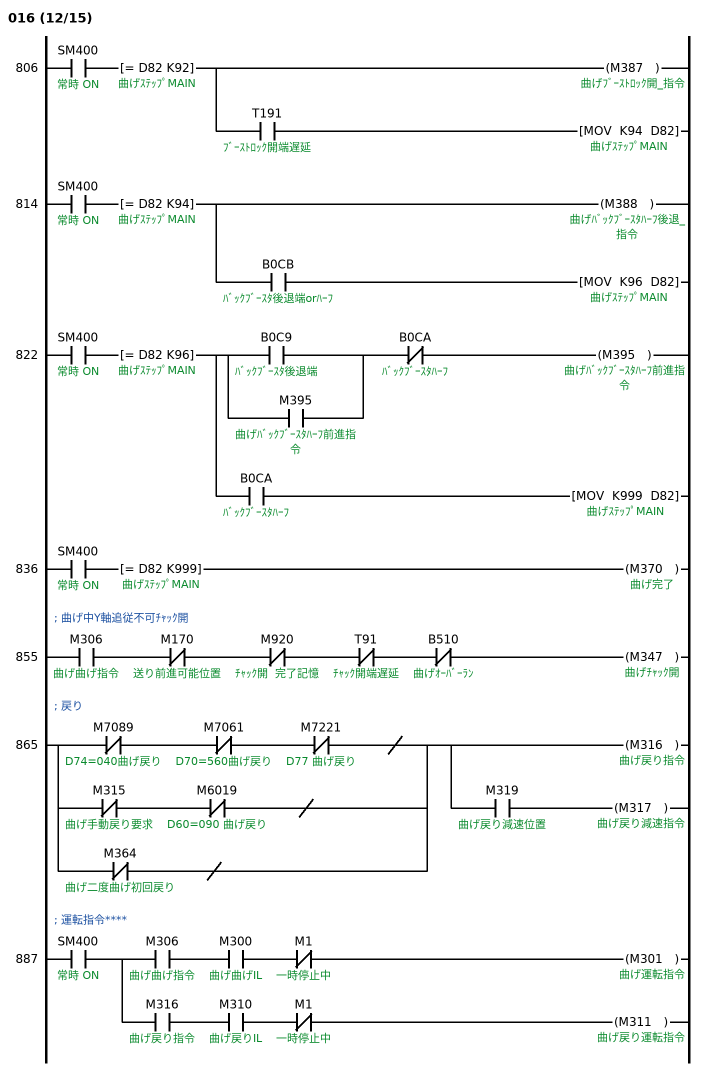
806   LD      SM400  ; 常時 ON
      AND=    D82 K92  ; 曲げｽﾃｯﾌﾟMAIN
      OUT     M387  ; 曲げﾌﾞｰｽﾄﾛｯｸ開_指令
      AND     T191  ; ﾌﾞｰｽﾄﾛｯｸ開端遅延
      MOV     K94 D82
814   LD      SM400  ; 常時 ON
      AND=    D82 K94  ; 曲げｽﾃｯﾌﾟMAIN
      OUT     M388  ; 曲げﾊﾞｯｸﾌﾞｰｽﾀﾊｰﾌ後退_指令
      AND     B0CB  ; ﾊﾞｯｸﾌﾞｰｽﾀ後退端orﾊｰﾌ
      MOV     K96 D82
822   LD      SM400  ; 常時 ON
      AND=    D82 K96  ; 曲げｽﾃｯﾌﾟMAIN
      MPS
      LD      B0C9  ; ﾊﾞｯｸﾌﾞｰｽﾀ後退端
      OR      M395  ; 曲げﾊﾞｯｸﾌﾞｰｽﾀﾊｰﾌ前進指令
      ANB
      ANI     B0CA  ; ﾊﾞｯｸﾌﾞｰｽﾀﾊｰﾌ
      OUT     M395  ; 曲げﾊﾞｯｸﾌﾞｰｽﾀﾊｰﾌ前進指令
      MPP
      AND     B0CA  ; ﾊﾞｯｸﾌﾞｰｽﾀﾊｰﾌ
      MOV     K999 D82
836   LD      SM400  ; 常時 ON
      AND=    D82 K999  ; 曲げｽﾃｯﾌﾟMAIN
      OUT     M370  ; 曲げ完了
; 曲げ中Y軸追従不可ﾁｬｯｸ開
855   LD      M306  ; 曲げ曲げ指令
      ANI     M170  ; 送り前進可能位置
      ANI     M920  ; ﾁｬｯｸ開  完了記憶
      ANI     T91  ; ﾁｬｯｸ開端遅延
      ANI     B510  ; 曲げｵｰﾊﾞｰﾗﾝ
      OUT     M347  ; 曲げﾁｬｯｸ開
; 戻り
865   LDI     M7089  ; D74=040曲げ戻り
      ANI     M7061  ; D70=560曲げ戻り
      ANI     M7221  ; D77 曲げ戻り
      INV
      LDI     M315  ; 曲げ手動戻り要求
      ANI     M6019  ; D60=090 曲げ戻り
      INV
      ORB
      LDI     M364  ; 曲げ二度曲げ初回戻り
      INV
      ORB
      OUT     M316  ; 曲げ戻り指令
      AND     M319  ; 曲げ戻り減速位置
      OUT     M317  ; 曲げ戻り減速指令
; 運転指令****
887   LD      SM400  ; 常時 ON
      MPS
      AND     M306  ; 曲げ曲げ指令
      AND     M300  ; 曲げ曲げIL
      ANI     M1  ; 一時停止中
      OUT     M301  ; 曲げ運転指令
      MPP
      AND     M316  ; 曲げ戻り指令
      AND     M310  ; 曲げ戻りIL
      ANI     M1  ; 一時停止中
      OUT     M311  ; 曲げ戻り運転指令
; 
      P1610
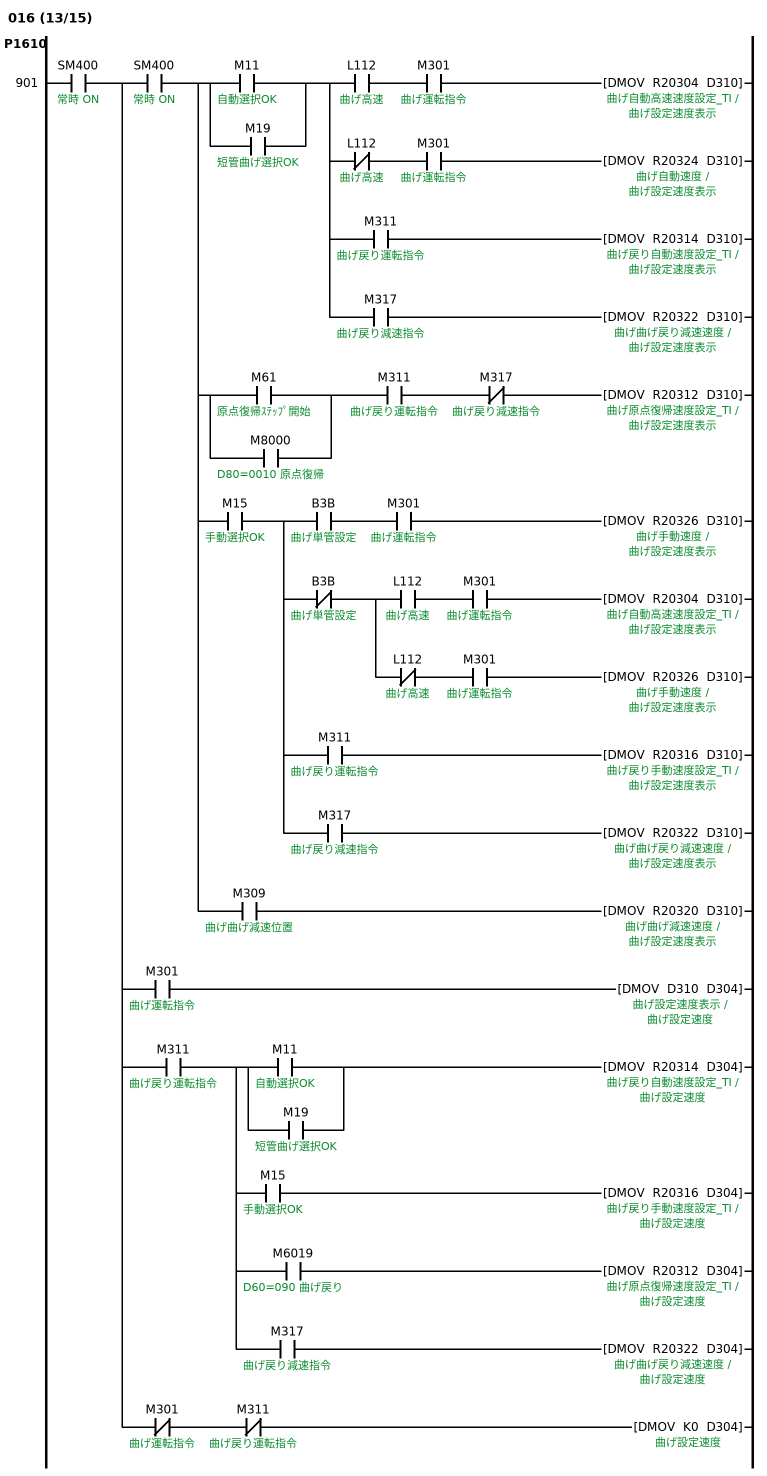
901   LD      SM400  ; 常時 ON
      MPS
      AND     SM400  ; 常時 ON
      MPS
      LD      M11  ; 自動選択OK
      OR      M19  ; 短管曲げ選択OK
      ANB
      MPS
      AND     L112  ; 曲げ高速
      AND     M301  ; 曲げ運転指令
      DMOV    R20304 D310  ; 曲げ自動高速速度設定_TI / 曲げ設定速度表示
      MRD
      ANI     L112  ; 曲げ高速
      AND     M301  ; 曲げ運転指令
      DMOV    R20324 D310  ; 曲げ自動速度
      MRD
      AND     M311  ; 曲げ戻り運転指令
      DMOV    R20314 D310  ; 曲げ戻り自動速度設定_TI
      MPP
      AND     M317  ; 曲げ戻り減速指令
      DMOV    R20322 D310  ; 曲げ曲げ戻り減速速度
      MRD
      LD      M61  ; 原点復帰ｽﾃｯﾌﾟ開始
      OR      M8000  ; D80=0010 原点復帰
      ANB
      AND     M311  ; 曲げ戻り運転指令
      ANI     M317  ; 曲げ戻り減速指令
      DMOV    R20312 D310  ; 曲げ原点復帰速度設定_TI
      MRD
      AND     M15  ; 手動選択OK
      MPS
      AND     B3B  ; 曲げ単管設定
      AND     M301  ; 曲げ運転指令
      DMOV    R20326 D310  ; 曲げ手動速度
      MRD
      ANI     B3B  ; 曲げ単管設定
      MPS
      AND     L112  ; 曲げ高速
      AND     M301  ; 曲げ運転指令
      DMOV    R20304 D310
      MPP
      ANI     L112  ; 曲げ高速
      AND     M301  ; 曲げ運転指令
      DMOV    R20326 D310
      MRD
      AND     M311  ; 曲げ戻り運転指令
      DMOV    R20316 D310  ; 曲げ戻り手動速度設定_TI
      MPP
      AND     M317  ; 曲げ戻り減速指令
      DMOV    R20322 D310
      MPP
      AND     M309  ; 曲げ曲げ減速位置
      DMOV    R20320 D310  ; 曲げ曲げ減速速度
      MRD
      AND     M301  ; 曲げ運転指令
      DMOV    D310 D304  ; 曲げ設定速度
      MRD
      AND     M311  ; 曲げ戻り運転指令
      MPS
      LD      M11  ; 自動選択OK
      OR      M19  ; 短管曲げ選択OK
      ANB
      DMOV    R20314 D304
      MRD
      AND     M15  ; 手動選択OK
      DMOV    R20316 D304
      MRD
      AND     M6019  ; D60=090 曲げ戻り
      DMOV    R20312 D304
      MPP
      AND     M317  ; 曲げ戻り減速指令
      DMOV    R20322 D304
      MPP
      ANI     M301  ; 曲げ運転指令
      ANI     M311  ; 曲げ戻り運転指令
      DMOV    K0 D304
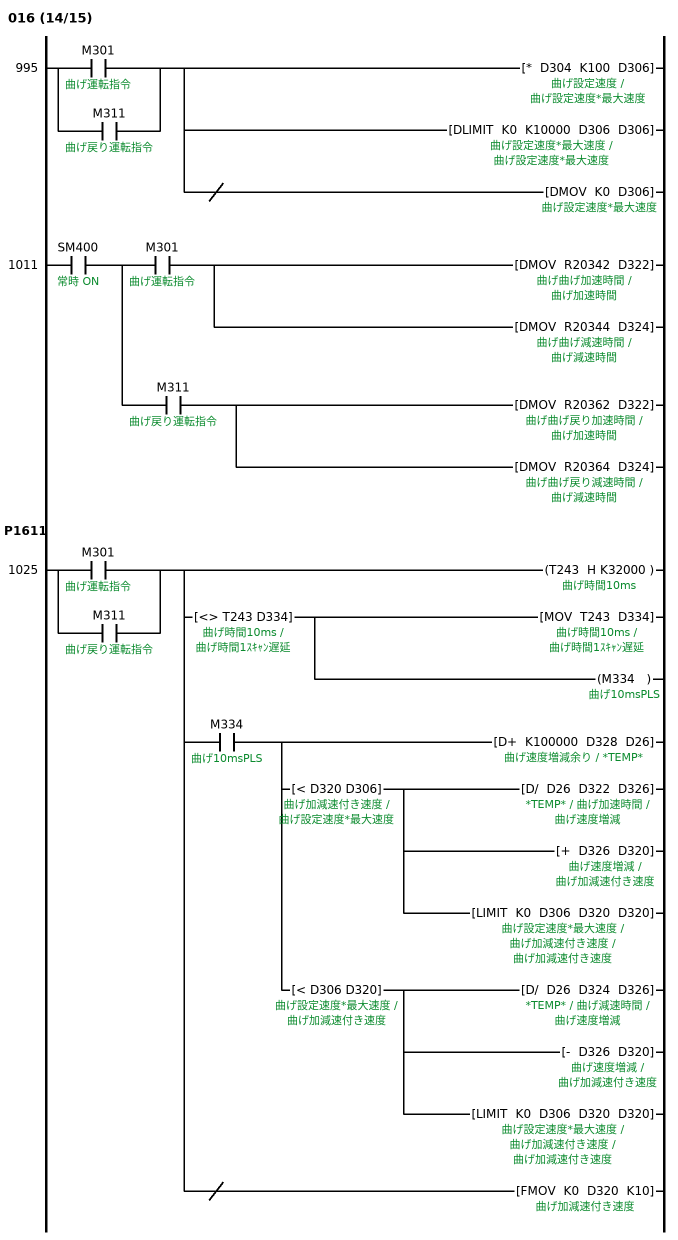
995   LD      M301  ; 曲げ運転指令
      OR      M311  ; 曲げ戻り運転指令
      *       D304 K100 D306  ; 曲げ設定速度*最大速度
      DLIMIT  K0 K10000 D306 D306
      INV
      DMOV    K0 D306
1011  LD      SM400  ; 常時 ON
      MPS
      AND     M301  ; 曲げ運転指令
      DMOV    R20342 D322  ; 曲げ曲げ加速時間 / 曲げ加速時間
      DMOV    R20344 D324  ; 曲げ曲げ減速時間 / 曲げ減速時間
      MPP
      AND     M311  ; 曲げ戻り運転指令
      DMOV    R20362 D322  ; 曲げ曲げ戻り加速時間
      DMOV    R20364 D324  ; 曲げ曲げ戻り減速時間
      P1611
1025  LD      M301  ; 曲げ運転指令
      OR      M311  ; 曲げ戻り運転指令
      OUTH    T243 K32000  ; 曲げ時間10ms
      MPS
      AND<>   T243 D334  ; 曲げ時間10ms / 曲げ時間1ｽｷｬﾝ遅延
      MOV     T243 D334
      OUT     M334  ; 曲げ10msPLS
      MRD
      AND     M334  ; 曲げ10msPLS
      D+      K100000 D328 D26  ; 曲げ速度増減余り
      MPS
      AND<    D320 D306  ; 曲げ加減速付き速度 / 曲げ設定速度*最大速度
      D/      D26 D322 D326  ; 曲げ速度増減
      +       D326 D320
      LIMIT   K0 D306 D320 D320
      MPP
      AND<    D306 D320  ; 曲げ設定速度*最大速度 / 曲げ加減速付き速度
      D/      D26 D324 D326
      -       D326 D320
      LIMIT   K0 D306 D320 D320
      MPP
      INV
      FMOV    K0 D320 K10
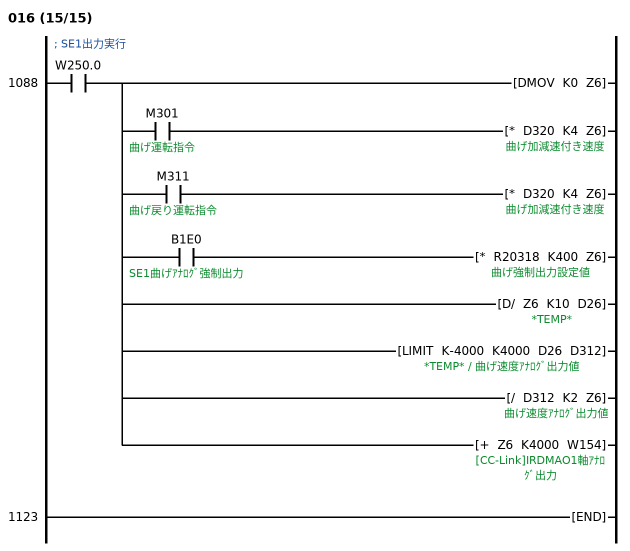
; SE1出力実行
1088  LD      W250.0
      DMOV    K0 Z6
      MPS
      AND     M301  ; 曲げ運転指令
      *       D320 K4 Z6
      MRD
      AND     M311  ; 曲げ戻り運転指令
      *       D320 K4 Z6
      MRD
      AND     B1E0  ; SE1曲げｱﾅﾛｸﾞ強制出力
      *       R20318 K400 Z6  ; 曲げ強制出力設定値
      MPP
      D/      Z6 K10 D26
      LIMIT   K-4000 K4000 D26 D312  ; 曲げ速度ｱﾅﾛｸﾞ出力値
      /       D312 K2 Z6
      +       Z6 K4000 W154  ; [CC-Link]IRDMAO1軸ｱﾅﾛｸﾞ出力
1123  END
END_PROGRAM

// device comments not shown above
R20951  ; PV2油圧制御値_X2#.#Mpa
R20961  ; PV2油圧測定値_Y2#.#Mpa
R20971  ; PV3油圧制御値_X2#.#Mpa
R20981  ; PV3油圧測定値_Y2#.#Mpa
R20991  ; PV4油圧制御値_X2#.#Mpa
R21001  ; PV4油圧測定値_Y2#.#Mpa
R22470  ; 曲げＲ1.5D
R22471  ; 曲げＲ2.0D
R23551  ; BT1_CP2
R23552  ; BT1_CP3
R23553  ; BT1_CP4
R23554  ; BT1_CP5
R23555  ; BT1_CP6
R23556  ; BT1_CP7
R23557  ; BT1_CP8
R23558  ; BT1_CP9
R23559  ; BT1_CP10
R23651  ; BT1_BP2
R23652  ; BT1_BP3
R23653  ; BT1_BP4
R23654  ; BT1_BP5
R23655  ; BT1_BP6
R23656  ; BT1_BP7
R23657  ; BT1_BP8
R23658  ; BT1_BP9
R23659  ; BT1_BP10
M63  ; ENC無原点位置OK
M77  ; 段取替機器ﾃﾞｰﾀ位置
M95  ; ﾊﾟｲﾌﾟ検出65A
M96  ; ﾊﾟｲﾌﾟ検出80A
M97  ; ﾊﾟｲﾌﾟ検出100A
M112  ; 送り手動後退条件
M146  ; 送り追従偏差警告減速
M147  ; 送り追従偏差小通常速
M173  ; 送り芯金受け干渉位置
M191  ; 送り1軸ｼｽﾃﾑﾋﾞｯﾄ異常完了
M196  ; 送り1軸原点ｼｽﾃﾑﾋﾞｯﾄ異常完了
M302  ; ﾍﾟﾝﾀﾞﾝﾄ曲げにて保持→寸動
M307  ; 曲げ曲げ減速指令
M312  ; 曲げ ﾍﾟﾝﾀﾞﾝﾄSW
M314  ; 曲げ戻り圧抜き指令
M363  ; 曲げ曲げ指令
M428  ; ｸﾗﾝﾌﾟﾀﾞｲ原点復帰完了
M704  ; ｸﾗﾝﾌﾟ無線_閉BS1ｽｷｬﾝ遅延
M714  ; ｸﾗﾝﾌﾟ無線_開BS1ｽｷｬﾝ遅延
M804  ; ﾌﾟﾚｯｼｬｰ無線_閉BS1ｽｷｬﾝ遅延
M814  ; ﾌﾟﾚｯｼｬｰ無線_開BS1ｽｷｬﾝ遅延
M924  ; ﾁｬｯｸ_圧選択_閉記憶一致
M956  ; ﾁｬｯｸ位置範囲O.K
M1006  ; 芯金ﾍﾟﾝﾀﾞﾝﾄ芯金前進
M1007  ; 芯金ﾍﾟﾝﾀﾞﾝﾄ芯金後退
M1100  ; ﾍｯﾄﾞｼﾌﾄR大右IL
M1103  ; ﾍｯﾄﾞｼﾌﾄ手動R大右進BS
M1104  ; ﾍｯﾄﾞｼﾌﾄ無線_R大右BS1ｽｷｬﾝ遅延
M1105  ; ﾍｯﾄﾞｼﾌﾄ手動R大右動作要求
M1110  ; ﾍｯﾄﾞｼﾌﾄR小左IL
M1113  ; ﾍｯﾄﾞｼﾌﾄ手動R小左BS
M1114  ; ﾍｯﾄﾞｼﾌﾄ無線_R小左BS1ｽｷｬﾝ遅延
M1115  ; ﾍｯﾄﾞｼﾌﾄ手動R小左動作要求
M1408  ; ﾌﾗﾝｼﾞ穴検出手動上昇自己保持
M1418  ; ﾌﾗﾝｼﾞ穴検出下降動作要求_自己保持
M1513  ; ﾜｲﾊﾟｰ注油手動注油BS
M1514  ; ﾜｲﾊﾟｰ注油手動注油開始指令
M1515  ; ﾜｲﾊﾟｰ注油手動注油開始要求
M1800  ; 端面検出端面検出IL
M1801  ; 端面検出端面検出開始
M1802  ; 端面検出端面検出記憶
M1803  ; 端面検出端面検出完了
M1805  ; 端面検出手動端面検出要求
M1820  ; 端面検出D88=010端面検出送り前進
M1821  ; 端面検出D88=020端面検出送り後退
M1822  ; 端面検出D88=010-20端面検出曲戻り
M1823  ; 端面検出D88=030端面検出ｴﾗｰ
M1824  ; 端面検出D88=***予備
M1825  ; 端面検出D89=***予備
M1826  ; 端面検出D90=***予備
M1827  ; 端面検出D88=999端面検出完了
M1921  ; ﾌﾗﾝｼﾞ穴検出D86=***_予備
M1926  ; ﾌﾗﾝｼﾞ穴検出D86=***_予備
M2128  ; ﾍﾞﾝﾄﾞﾍｯﾄﾞｼﾌﾄ原点復帰完了
M2401  ; ﾘﾄﾗｸﾄﾌﾟﾚｯｼｬｰ位置決め前進可能条件
M2508  ; ﾘﾄﾗｸﾄﾌﾟﾚｯｼｬｰ上下移動手動上昇自己
M2516  ; ﾘﾄﾗｸﾄﾌﾟﾚｯｼｬｰ上下移動下降ﾌﾗﾝｼﾞ検
M2518  ; ﾘﾄﾗｸﾄﾌﾟﾚｯｼｬｰ上下移動下降動作要求
M3003  ; 管外形　予備1
M3004  ; 管外形　予備2
M3005  ; 管外形　予備3
M3006  ; 管外形　予備4
M3201  ; ﾛｯﾄNo.-02作業完了
M3202  ; ﾛｯﾄNo.-03作業完了
M3203  ; ﾛｯﾄNo.-04作業完了
M3204  ; ﾛｯﾄNo.-05作業完了
M3205  ; ﾛｯﾄNo.-06作業完了
M3206  ; ﾛｯﾄNo.-07作業完了
M3207  ; ﾛｯﾄNo.-08作業完了
M3208  ; ﾛｯﾄNo.-09作業完了
M3209  ; ﾛｯﾄNo.-10作業完了
M3210  ; ﾛｯﾄNo.-11作業完了
M3211  ; ﾛｯﾄNo.-12作業完了
M3212  ; ﾛｯﾄNo.-13作業完了
M3213  ; ﾛｯﾄNo.-14作業完了
M3214  ; ﾛｯﾄNo.-15作業完了
M3215  ; ﾛｯﾄNo.-16作業完了
M3216  ; ﾛｯﾄNo.-17作業完了
M3217  ; ﾛｯﾄNo.-18作業完了
M3218  ; ﾛｯﾄNo.-19作業完了
M3219  ; ﾛｯﾄNo.-20作業完了
M3220  ; ﾛｯﾄNo.-21作業完了
M3221  ; ﾛｯﾄNo.-22作業完了
M3222  ; ﾛｯﾄNo.-23作業完了
M3223  ; ﾛｯﾄNo.-24作業完了
M3224  ; ﾛｯﾄNo.-25作業完了
M3225  ; ﾛｯﾄNo.-26作業完了
M3226  ; ﾛｯﾄNo.-27作業完了
M3227  ; ﾛｯﾄNo.-28作業完了
M3228  ; ﾛｯﾄNo.-29作業完了
M3229  ; ﾛｯﾄNo.-30作業完了
M3303  ; 次段管外形　予備1
M3304  ; 次段管外形　予備2
M3305  ; 次段管外形　予備3
M3306  ; 次段管外形　予備4
M5008  ; [TP]B008表示中
M5009  ; [TP]B009表示中
M5010  ; [TP]B010表示中
M5011  ; [TP]B011表示中
M5012  ; [TP]B012表示中
M5013  ; [TP]B013表示中
M5014  ; [TP]B014表示中
M5015  ; [TP]B015表示中
M5016  ; [TP]B016表示中
M5017  ; [TP]B017表示中
M5018  ; [TP]B018表示中
M5019  ; [TP]B019表示中
M5020  ; [TP]B020表示中
M5021  ; [TP]B021表示中
M5022  ; [TP]B022表示中
M5023  ; [TP]B023表示中
M5024  ; [TP]B024表示中
M5025  ; [TP]B025表示中
M5026  ; [TP]B026表示中
M5027  ; [TP]B027表示中
M5028  ; [TP]B028表示中
M5029  ; [TP]B029表示中
M5030  ; [TP]B030表示中
M5031  ; [TP]B031表示中
M5032  ; [TP]B032表示中
M5033  ; [TP]B033表示中
M5034  ; [TP]B034表示中
M5035  ; [TP]B035表示中
M5036  ; [TP]B036表示中
M5037  ; [TP]B037表示中
M5038  ; [TP]B038表示中
M5039  ; [TP]B039表示中
M5040  ; [TP]B040表示中
M5044  ; [TP]B044表示中
M5046  ; [TP]B046表示中
M5047  ; [TP]B047表示中
M5048  ; [TP]B048表示中
M5052  ; [TP]B052表示中
M5053  ; [TP]B053表示中
M5054  ; [TP]B054表示中
M5055  ; [TP]B055表示中
M5056  ; [TP]B056表示中
M5057  ; [TP]B057表示中
M5058  ; [TP]B058表示中
M5059  ; [TP]B059表示中
M5063  ; [TP]B063表示中
M5066  ; [TP]B066表示中
M5067  ; [TP]B067表示中
M5068  ; [TP]B068表示中
M5069  ; [TP]B069表示中
M5070  ; [TP]B070表示中
M5071  ; [TP]B071表示中
M5072  ; [TP]B072表示中
M5073  ; [TP]B073表示中
M5074  ; [TP]B074表示中
M5075  ; [TP]B075表示中
M5076  ; [TP]B076表示中
M5077  ; [TP]B077表示中
M5078  ; [TP]B078表示中
M5079  ; [TP]B079表示中
M5084  ; [TP]B084表示中
M5085  ; [TP]B085表示中
M5086  ; [TP]B086表示中
M5087  ; [TP]B087表示中
M5088  ; [TP]B088表示中
M5089  ; [TP]B089表示中
M5090  ; [TP]B090表示中
M5091  ; [TP]B091表示中
M5092  ; [TP]B092表示中
M5093  ; [TP]B093表示中
M5094  ; [TP]B094表示中
M5095  ; [TP]B095表示中
M5108  ; [TP]ｲﾝﾀｰﾛｯｸ画面
M5110  ; [TP]隠しﾊﾟﾗﾒｰﾀ画面
M5111  ; [TP]予備画面
M5113  ; [TP]ｱﾗｰﾑ画面緑点灯
M5114  ; [TP]ｱﾗｰﾑ画面赤点滅
M5121  ; [TP]B101表示
M5141  ; [TP]W41表示中
M5142  ; [TP]W42表示中
M5143  ; [TP]W43表示中
M5144  ; [TP]W44表示中
M5145  ; [TP]W45表示中
M5146  ; [TP]W46表示中
M5147  ; [TP]W47表示中
M5148  ; [TP]W48表示中
M5149  ; [TP]W49表示中
M5150  ; [TP]W50表示中
M5151  ; [TP]W51表示中
M5152  ; [TP]W52表示中
M5153  ; [TP]W53表示中
M5154  ; [TP]W54表示中
M5155  ; [TP]W55表示中
M5156  ; [TP]W56表示中
M5157  ; [TP]W57表示中
M5158  ; [TP]W58表示中
M5159  ; [TP]W59表示中
M5161  ; WIN1_W41表示中
M5162  ; WIN1_W42表示中
M5163  ; WIN1_W43表示中
M5164  ; WIN1_W44表示中
M5165  ; WIN1_W45表示中
M5166  ; WIN1_W46表示中
M5167  ; WIN1_W47表示中
M5168  ; WIN1_W48表示中
M5169  ; WIN1_W49表示中
M5170  ; WIN1_W50表示中
M5171  ; WIN1_W51表示中
M5172  ; WIN1_W52表示中
M5173  ; WIN1_W53表示中
M5174  ; WIN1_W54表示中
M5175  ; WIN1_W55表示中
M5176  ; WIN1_W56表示中
M5177  ; WIN1_W57表示中
M5178  ; WIN1_W58表示中
M5179  ; WIN1_W59表示中
M5181  ; WIN2_W41表示中
M5182  ; WIN2_W42表示中
M5183  ; WIN2_W43表示中
M5184  ; WIN2_W44表示中
M5185  ; WIN2_W45表示中
M5186  ; WIN2_W46表示中
M5187  ; WIN2_W47表示中
M5188  ; WIN2_W48表示中
M5189  ; WIN2_W49表示中
M5190  ; WIN2_W50表示中
M5191  ; WIN2_W51表示中
M5192  ; WIN2_W52表示中
M5193  ; WIN2_W53表示中
M5194  ; WIN2_W54表示中
M5195  ; WIN2_W55表示中
M5196  ; WIN2_W56表示中
M5197  ; WIN2_W57表示中
M5198  ; WIN2_W58表示中
M5199  ; WIN2_W59表示中
M5205  ; 異常検出記憶
M5210  ; ﾃﾞｰﾀ要求
M5232  ; 全製品完IL
M5300  ; 40Aﾘﾓｰﾄﾃﾞｰﾀ
M5301  ; 50Aﾘﾓｰﾄﾃﾞｰﾀ
M5302  ; 65Aﾘﾓｰﾄﾃﾞｰﾀ
M5303  ; 80Aﾘﾓｰﾄﾃﾞｰﾀ
M5304  ; 100Aﾘﾓｰﾄﾃﾞｰﾀ
M5310  ; ﾌﾗﾝｼﾞﾁｬｯｸ側5K_ﾘﾓｰﾄﾃﾞｰﾀ
M5311  ; ﾌﾗﾝｼﾞﾁｬｯｸ側10K_ﾘﾓｰﾄﾃﾞｰﾀ
M5312  ; ﾌﾗﾝｼﾞﾁｬｯｸ側16K_ﾘﾓｰﾄﾃﾞｰﾀ
M5313  ; ﾌﾗﾝｼﾞﾁｬｯｸ側20K_ﾘﾓｰﾄﾃﾞｰﾀ
M5314  ; ﾌﾗﾝｼﾞﾁｬｯｸ側30K_ﾘﾓｰﾄﾃﾞｰﾀ
M6021  ; D60=120 ﾍｯﾄﾞｼﾌﾄ原点ｾｯﾄ
M6022  ; D60=86
M6024  ; ｷｬﾚｯｼﾞ原点復帰
M6029  ; ﾍｯﾄﾞｼﾌﾄ原点復帰
M7001  ; D70=010ﾊﾟｲﾌﾟ受け上昇(未使用)
M7015  ; D70=150予備
M7018  ; D70=180
M7034  ; D70=231ﾌﾟﾚｯｼｬ台前進(未使用)
M7036  ; D70=
M7037  ; D70=
M7044  ; D70=231ﾌﾟﾚｯｼｬ台前進端異常
M7060  ; D70=550搬出完了
M7062  ; D70=570予備
M7069  ; D70=640
M7070  ; D70=650
M7071  ; D70=660
M7072  ; D70=670
M7073  ; D70=680
M7096  ; D74=060予備
M7102  ; D75=999ｷｬﾚｯｼﾞ退避完了
L66  ; ﾛｯﾄ№-02作業完了記憶
L67  ; ﾛｯﾄ№-03作業完了記憶
L68  ; ﾛｯﾄ№-04作業完了記憶
L69  ; ﾛｯﾄ№-05作業完了記憶
L70  ; ﾛｯﾄ№-06作業完了記憶
L71  ; ﾛｯﾄ№-07作業完了記憶
L72  ; ﾛｯﾄ№-08作業完了記憶
L73  ; ﾛｯﾄ№-09作業完了記憶
L74  ; ﾛｯﾄ№-10作業完了記憶
L75  ; ﾛｯﾄ№-11作業完了記憶
L76  ; ﾛｯﾄ№-12作業完了記憶
L77  ; ﾛｯﾄ№-13作業完了記憶
L78  ; ﾛｯﾄ№-14作業完了記憶
L79  ; ﾛｯﾄ№-15作業完了記憶
L80  ; ﾛｯﾄ№-16作業完了記憶
L81  ; ﾛｯﾄ№-17作業完了記憶
L82  ; ﾛｯﾄ№-18作業完了記憶
L83  ; ﾛｯﾄ№-19作業完了記憶
L84  ; ﾛｯﾄ№-20作業完了記憶
L85  ; ﾛｯﾄ№-21作業完了記憶
L86  ; ﾛｯﾄ№-22作業完了記憶
L87  ; ﾛｯﾄ№-23作業完了記憶
L88  ; ﾛｯﾄ№-24作業完了記憶
L89  ; ﾛｯﾄ№-25作業完了記憶
L90  ; ﾛｯﾄ№-26作業完了記憶
L91  ; ﾛｯﾄ№-27作業完了記憶
L92  ; ﾛｯﾄ№-28作業完了記憶
L93  ; ﾛｯﾄ№-29作業完了記憶
L94  ; ﾛｯﾄ№-30作業完了記憶
L115  ; ペンダント無
L119  ; 芯金微調整_ﾌﾟﾘｾｯﾄ有_TB
L124  ; ﾍｯﾄﾞｼﾌﾄ_ﾌﾟﾘｾｯﾄ有_TB
L125  ; 芯金横移動_ﾌﾟﾘｾｯﾄ有_TB
L129  ; ｺﾒﾝﾄ有_TB
L132  ; 省略手動選択_TB
L154  ; ｱｼﾞﾃｰｼｮﾝ_無選択
L155  ; ｱｼﾞﾃｰｼｮﾝ_有選択
L2111  ; 40A選択 ﾗﾝﾌﾟON
L2112  ; 50A選択 ﾗﾝﾌﾟON
L2113  ; 65A選択 ﾗﾝﾌﾟON
L2114  ; 80A選択 ﾗﾝﾌﾟON
L2115  ; 100A選択ﾗﾝﾌﾟON
L2116  ; SGP     ﾗﾝﾌﾟON
L2117  ; #40     ﾗﾝﾌﾟON
L2118  ; #80     ﾗﾝﾌﾟON
L2119  ; #160    ﾗﾝﾌﾟON
L2120  ; E管選択 ﾗﾝﾌﾟON
L2121  ; S管選択 ﾗﾝﾌﾟON
L2122  ; 穴検ﾓｰﾄﾞ自動ﾗﾝﾌﾟON
L2123  ; 穴検ﾓｰﾄﾞ 手動ﾗﾝﾌﾟON
L2124  ; 穴検ﾓｰﾄﾞ無ﾗﾝﾌﾟON
L2125  ; ｽﾘｰﾌﾞ選択有ﾗﾝﾌﾟON
L2126  ; ｽﾘｰﾌﾞ選択無ﾗﾝﾌﾟON
L2250  ; ﾁｬｯｸ側素管ﾗﾝﾌﾟON
L2251  ; ﾁｬｯｸ側ﾌﾗﾝｼﾞﾗﾝﾌﾟON
L2252  ; ﾁｬｯｸ側ｽﾘｰﾌﾞﾗﾝﾌﾟON
L2254  ; 曲げ側素管ﾗﾝﾌﾟON
L2255  ; 曲げ側ﾌﾗﾝｼﾞﾗﾝﾌﾟON
L2256  ; 曲げ側ｽﾘｰﾌﾞﾗﾝﾌﾟON
L2260  ; ﾌﾗﾝｼﾞ 5k ﾗﾝﾌﾟON
L2261  ; ﾌﾗﾝｼﾞ 10k ﾗﾝﾌﾟON
L2262  ; ﾌﾗﾝｼﾞ 16k ﾗﾝﾌﾟON
X1  ; CC_LINK ﾃﾞｰﾀﾘﾝｸ中
X0F  ; CC_LINK UNIT_READY
X4A  ; ﾎﾟﾝﾌﾟMC ON
X61  ; ｵｲﾙｺﾝ　異常ﾚﾍﾞﾙ
X0E4  ; 軸1MｺｰﾄﾞON(送り)
X0E5  ; 軸2MｺｰﾄﾞON
X0E9  ; 軸2ｴﾗｰ検出
X0ED  ; 軸2BUSY()
X0F0  ; 軸1始動完了(送り)
X0F1  ; 軸2始動完了()
X0F5  ; 軸2位置決め完了()
X159A  ; IRDM-CCLｴﾗｰ状態
Y0E5  ; 軸2軸停止()
Y0E8  ; 軸1正転JOG始動(送り)
Y0E9  ; 軸1逆転JOG始動(送り)
Y0EA  ; 軸2正転JOG始動()
Y0EB  ; 軸2逆転JOG始動()
Y0F0  ; 軸1位置決め始動(送り)
Y0F1  ; 軸2位置決め始動()
Y0F4  ; 軸1実行禁止ﾌﾗｸﾞ(送り)
Y0F5  ; 軸2実行禁止ﾌﾗｸﾞ()
Y1190  ; ｸﾗﾝﾌﾟﾀﾞｲ P1一致信号ﾘｾｯﾄ指令
Y1192  ; ｸﾗﾝﾌﾟﾀﾞｲ 一致信号ｲﾈｰﾌﾞﾙ
Y1193  ; ｸﾗﾝﾌﾟﾀﾞｲ 減算ｶｳﾝﾄ指令
Y1196  ; ｸﾗﾝﾌﾟﾀﾞｲ ｶｳﾝﾀ機能選択開始指令
Y1197  ; ﾌﾟﾚｯｼｬﾀﾞｲ P1一致信号ﾘｾｯﾄ指令
Y1199  ; ﾌﾟﾚｯｼｬﾀﾞｲ 一致信号ｲﾈｰﾌﾞﾙ
Y119A  ; ﾌﾟﾚｯｼｬﾀﾞｲ 減算ｶｳﾝﾄ指令
Y119D  ; ﾌﾟﾚｯｼｬﾀﾞｲ ｶｳﾝﾀ機能選択開始指令
Y11A0  ; ｸﾗﾝﾌﾟﾀﾞｲ 外部ﾌﾟﾘｾｯﾄ検出ﾘｾｯﾄ指令
Y11A1  ; ｸﾗﾝﾌﾟﾀﾞｲ P2一致信号ﾘｾｯﾄ指令
Y11A2  ; ﾌﾟﾚｯｼｬﾀﾞｲ 外部ﾌﾟﾘｾｯﾄ検出ﾘｾｯﾄ指令
Y11A3  ; ﾌﾟﾚｯｼｬﾀﾞｲ P2一致信号ﾘｾｯﾄ指令
Y1210  ; 曲げ P1一致信号ﾘｾｯﾄ指令
Y1212  ; 曲げ 一致信号ｲﾈｰﾌﾞﾙ
Y1213  ; 曲げ 減算ｶｳﾝﾄ指令
Y1216  ; 曲げ ｶｳﾝﾀ機能選択開始指令
Y1217  ; ﾍﾞﾝﾄﾞﾍｯﾄﾞｼﾌﾄ P1一致信号ﾘｾｯﾄ指令
Y1219  ; ﾍﾞﾝﾄﾞﾍｯﾄﾞｼﾌﾄ 一致信号ｲﾈｰﾌﾞﾙ
Y121A  ; ﾍﾞﾝﾄﾞﾍｯﾄﾞｼﾌﾄ 減算ｶｳﾝﾄ指令
Y121D  ; ﾍﾞﾝﾄﾞﾍｯﾄﾞｼﾌﾄ ｶｳﾝﾀ機能選択開始指
Y1220  ; 曲げ 外部ﾌﾟﾘｾｯﾄ検出ﾘｾｯﾄ指令
Y1221  ; 曲げ P2一致信号ﾘｾｯﾄ指令
Y1222  ; ﾍﾞﾝﾄﾞﾍｯﾄﾞｼﾌﾄ 外部ﾌﾟﾘｾｯﾄ検出ﾘｾｯﾄ
Y1223  ; ﾍﾞﾝﾄﾞﾍｯﾄﾞｼﾌﾄ P2一致信号ﾘｾｯﾄ指令
Y1290  ; ﾋﾈﾘ P1一致信号ﾘｾｯﾄ指令
Y1292  ; ﾋﾈﾘ 一致信号ｲﾈｰﾌﾞﾙ
Y1293  ; ﾋﾈﾘ 減算ｶｳﾝﾄ指令
Y1296  ; ﾋﾈﾘ ｶｳﾝﾀ機能選択開始指令
Y1297  ; ﾁｬｯｸ開/閉 P1一致信号ﾘｾｯﾄ指令
Y1299  ; ﾁｬｯｸ開/閉 一致信号ｲﾈｰﾌﾞﾙ
Y129A  ; ﾁｬｯｸ開/閉 減算ｶｳﾝﾄ指令
Y129D  ; ﾁｬｯｸ開/閉 ｶｳﾝﾀ機能選択開始指令
Y12A0  ; ﾋﾈﾘ 外部ﾌﾟﾘｾｯﾄ検出ﾘｾｯﾄ指令
Y12A1  ; ﾋﾈﾘ P2一致信号ﾘｾｯﾄ指令
Y12A2  ; ﾁｬｯｸ開/閉 外部ﾌﾟﾘｾｯﾄ検出ﾘｾｯﾄ指令
Y12A3  ; ﾁｬｯｸ開/閉 P2一致信号ﾘｾｯﾄ指令
Y13C6  ; SV21 ﾁｬｯｸ 閉（Wup圧）
Y159A  ; IRDM-CCLｴﾗｰﾘｾｯﾄ要求
B6  ; ｳｫｰﾐｲﾝｸﾞｱｯﾌﾟ完了_仮設TB
B8  ; ENTｷｰ
B9F  ; ﾁｬｯｸ原点復帰完了記憶
B0EA  ; ﾘﾄﾗｸﾄﾌﾟﾚｯｼｬ有
B0F4  ; ﾊﾟｽﾜｰﾄﾞ変更_TB
B0F5  ; ﾊﾟｽﾜｰﾄﾞ書換_TB
B0FD  ; ｲﾝﾀｰﾛｯｸ解除_TB
B12B  ; ﾘﾄﾗｸﾄﾌﾟﾚｯｼｬ自動準備
B14C  ; 手動穴検_正転TB
B14D  ; 手動穴検_逆転TB
B18A  ; ﾘﾄﾗｸﾄﾌﾟﾚｯｼｬﾛｯｸ有
B1B6  ; SV21ﾊﾟｲﾌﾟﾁｬｯｸ
B1B7  ; SV22ﾊﾟｲﾌﾟﾁｬｯｸ
B204  ; B20_ﾃﾞｰﾀ変換_TB
B205  ; B20_ﾃﾞｰﾀｸﾘｱ_TB
B207  ; ｲｰﾄﾝ式
B227  ; ﾜｰｸ選択SWﾋﾞｯﾄ
B233  ; ﾜｰｸﾃﾞｰﾀ変換_TB
B251  ; B3_ST02点滅
B252  ; B3_ST03点滅
B253  ; B3_ST04点滅
B254  ; B3_ST05点滅
B255  ; B3_ST06点滅
B256  ; B3_ST07点滅
B257  ; B3_ST08点滅
B258  ; B3_ST09点滅
B259  ; B3_ST10点滅
B25A  ; B3_ST11点滅
B280  ; B98_ST01緑表示
B281  ; B98_ST02緑表示
B282  ; B98_ST03緑表示
B283  ; B98_ST04緑表示
B284  ; B98_ST05緑表示
B285  ; B98_ST06緑表示
B286  ; B98_ST07緑表示
B287  ; B98_ST08緑表示
B288  ; B98_ST09緑表示
B289  ; B98_ST10緑表示
B313  ; 曲げ速度高速選択
B314  ; 終点ﾌﾗﾝｼﾞ有
B315  ; 視点ﾌﾗﾝｼﾞ有
B32B  ; #160選択
B349  ; ﾌﾗﾝｼﾞ 10k ﾗﾝﾌﾟON
B34A  ; ﾌﾗﾝｼﾞ 16k ﾗﾝﾌﾟON
B34B  ; ﾌﾗﾝｼﾞ 20k ﾗﾝﾌﾟON
B34C  ; ﾌﾗﾝｼﾞ 30k ﾗﾝﾌﾟON
B900  ; ﾘﾄﾗｸﾄﾌﾟﾚｯｼｬﾛｯｸ閉_TB
B901  ; ﾘﾄﾗｸﾄﾌﾟﾚｯｼｬﾛｯｸ開_TB
B903  ; ﾘﾄﾗｸﾄﾌﾟﾚｯｼｬﾛｯｸ閉_TL
B904  ; ﾘﾄﾗｸﾄﾌﾟﾚｯｼｬﾛｯｸ開_TL
B905  ; ﾘﾄﾗｸﾄﾌﾟﾚｯｼｬﾛｯｸ運転中
B906  ; ﾘﾄﾗｸﾄﾌﾟﾚｯｼｬﾛｯｸ閉_可TL
B907  ; ﾘﾄﾗｸﾄﾌﾟﾚｯｼｬﾛｯｸ開_可TL
B908  ; ﾘﾄﾗｸﾄﾌﾟﾚｯｼｬﾛｯｸ閉端
B909  ; ﾘﾄﾗｸﾄﾌﾟﾚｯｼｬﾛｯｸ開端
B90A  ; ﾘﾄﾗｸﾄﾌﾟﾚｯｼｬﾛｯｸ有
D11  ; 書込中 to PLC
D12  ; 書込完了 to PLC
D27  ; *TEMP*
D29  ; *TEMP*
D72  ; 自動運転ｽﾃｯﾌﾟSUB2
D85  ; 曲げ戻りｽﾃｯﾌﾟMAIN
D88  ; 端面検出ｽﾃｯﾌﾟ
D118  ; 送りﾄﾙｸ制限出力値
D124  ; 送り偏差回転数
D126  ; 送りmm
D142  ; 送り検出後送り位置記憶
D160  ; 送り TEMP
D169  ; 送りMd102(852)偏差ｶｳﾝﾀ
D179  ; 送りMd103(855)
D191  ; 送り1-1軸完了ｽﾃｰﾀｽ
D196  ; 送り1-1軸原点完了ｽﾃｰﾀｽ
D252  ; ﾋﾈﾘ今回目標移動量表示
D332  ; 曲げYn+1設定角度
D362  ; 曲げﾘﾄﾗｸﾄ判断用曲げ周長
D622  ; ﾁｬｯｸ前ｽｷｬﾝ現在値
D626  ; ﾁｬｯｸ登録値
D750  ; SE4_設定値
D760  ; SE1_設定値
D768  ; SE1_出力値
D812  ; ｽﾘｰﾌﾞﾛﾝｸﾞ
D814  ; ｽﾘｰﾌﾞﾐﾄﾞﾙ
D816  ; ｽﾘｰﾌﾞｼｮｰﾄ
D1000  ; ｻｲﾄﾞﾌﾞｰｽﾀｰ現在値
D1002  ; ｻｲﾄﾞﾌﾞｰｽﾀｰ前ｽｷｬﾝ現在値
D1004  ; ｻｲﾄﾞﾌﾞｰｽﾀｰ設定速度
D1006  ; ｻｲﾄﾞﾌﾞｰｽﾀｰ設定速度*最大速度
D1010  ; ｻｲﾄﾞﾌﾞｰｽﾀｰ設定速度表示
D1012  ; ｻｲﾄﾞﾌﾞｰｽﾀｰ速度ｱﾅﾛｸﾞ出力値
D1020  ; ｻｲﾄﾞﾌﾞｰｽﾀｰ加減速付き速度
D1022  ; ｻｲﾄﾞﾌﾞｰｽﾀｰ加速時間
D1024  ; ｻｲﾄﾞﾌﾞｰｽﾀｰ減速時間
D1026  ; ｻｲﾄﾞﾌﾞｰｽﾀｰ速度増減
D1028  ; ｻｲﾄﾞﾌﾞｰｽﾀｰ速度増減余り
D1030  ; ｻｲﾄﾞﾌﾞｰｽﾀｰ自動設定角度
D1032  ; ｻｲﾄﾞﾌﾞｰｽﾀｰYn+1設定角度
D1034  ; ｻｲﾄﾞﾌﾞｰｽﾀｰ時間1ｽｷｬﾝ遅延
D1040  ; ｻｲﾄﾞﾌﾞｰｽﾀｰ目標値
D1042  ; ｻｲﾄﾞﾌﾞｰｽﾀｰ曲げ停止位置
D1044  ; ｻｲﾄﾞﾌﾞｰｽﾀｰ戻り停止位置
D1046  ; ｻｲﾄﾞﾌﾞｰｽﾀｰ曲げ減速位置
D1048  ; ｻｲﾄﾞﾌﾞｰｽﾀｰ戻り減速位置
D1201  ; B25表示_ST点滅判定用
D1212  ; B25表示_Y2mm
D1214  ; B25表示_Y3mm
D1216  ; B25表示_Y4mm
D1218  ; B25表示_Y5mm
D1220  ; B25表示_Y6mm
D1222  ; B25表示_Y7mm
D1224  ; B25表示_Y8mm
D1226  ; B25表示_Y9mm
D1228  ; B25表示_Y10mm
D1230  ; B25表示_Y11mm
D1242  ; B25表示_B2°
D1244  ; B25表示_B3°
D1246  ; B25表示_B4°
D1248  ; B25表示_B5°
D1250  ; B25表示_B6°
D1252  ; B25表示_B7°
D1254  ; B25表示_B8°
D1256  ; B25表示_B9°
D1258  ; B25表示_B10°
D1270  ; B25表示_C1°
D1272  ; B25表示_C2°
D1274  ; B25表示_C3°
D1276  ; B25表示_C4°
D1278  ; B25表示_C5°
D1280  ; B25表示_C6°
D1282  ; B25表示_C7°
D1284  ; B25表示_C8°
D1286  ; B25表示_C9°
D1288  ; B25表示_C10°
D1290  ; B25表示_C11°
D1412  ; B43入力_YM2mm
D1414  ; B43入力_YM3mm
D1416  ; B43入力_YM4mm
D1418  ; B43入力_YM5mm
D1420  ; B43入力_YM6mm
D1422  ; B43入力_YM7mm
D1424  ; B43入力_YM8mm
D1426  ; B43入力_YM9mm
D1428  ; B43入力_YM10mm
D1430  ; B43入力_YM11mm
D1442  ; B43入力_BM2°
D1444  ; B43入力_BM3°
D1446  ; B43入力_BM4°
D1448  ; B43入力_BM5°
D1450  ; B43入力_BM6°
D1452  ; B43入力_BM7°
D1454  ; B43入力_BM8°
D1456  ; B43入力_BM9°
D1458  ; B43入力_BM10°
D1460  ; B43入力_BM11°
D1472  ; B43入力_CM2°
D1474  ; B43入力_CM3°
D1476  ; B43入力_CM4°
D1478  ; B43入力_CM5°
D1480  ; B43入力_CM6°
D1482  ; B43入力_CM7°
D1484  ; B43入力_CM8°
D1486  ; B43入力_CM9°
D1488  ; B43入力_CM10°
D1490  ; B43入力_CM11°
D1512  ; B43入力_YM2mm
D1514  ; B43入力_YM3mm
D1516  ; B43入力_YM4mm
D1518  ; B43入力_YM5mm
D1520  ; B43入力_YM6mm
D1522  ; B43入力_YM7mm
D1524  ; B43入力_YM8mm
D1526  ; B43入力_YM9mm
D1528  ; B43入力_YM10mm
D1530  ; B43入力_YM11mm
D1542  ; B43入力_BM2°
D1544  ; B43入力_BM3°
D1546  ; B43入力_BM4°
D1548  ; B43入力_BM5°
D1550  ; B43入力_BM6°
D1552  ; B43入力_BM7°
D1554  ; B43入力_BM8°
D1556  ; B43入力_BM9°
D1558  ; B43入力_BM10°
D1560  ; B43入力_BM11°
D1572  ; B43入力_CM2°
D1574  ; B43入力_CM3°
D1576  ; B43入力_CM4°
D1578  ; B43入力_CM5°
D1580  ; B43入力_CM6°
D1582  ; B43入力_CM7°
D1584  ; B43入力_CM8°
D1586  ; B43入力_CM9°
D1588  ; B43入力_CM10°
D1590  ; B43入力_CM11°
D1601  ; B43入力_BT2
D1602  ; B43入力_BT3
D1603  ; B43入力_BT4
D1604  ; B43入力_BT5
D1605  ; B43入力_BT6
D1606  ; B43入力_BT7
D1607  ; B43入力_BT8
D1608  ; B43入力_BT9
D1609  ; B43入力_BT10
D1610  ; B43入力_BT11
D2000  ; W50表示01行目  ﾊﾟｰﾂ№  1/8
D2001  ; W50表示01行目  ﾊﾟｰﾂ№  2/8
D2002  ; W50表示01行目  ﾊﾟｰﾂ№  3/8
D2003  ; W50表示01行目  ﾊﾟｰﾂ№  4/8
D2004  ; W50表示01行目  ﾊﾟｰﾂ№  5/8
D2005  ; W50表示01行目  ﾊﾟｰﾂ№  6/8
D2006  ; W50表示01行目  ﾊﾟｰﾂ№  7/8
D2007  ; W50表示01行目  ﾊﾟｰﾂ№  8/8
D2008  ; W50表示01行目  予備1   1/6
D2009  ; W50表示01行目  予備1   2/6
D2010  ; W50表示01行目  予備1   3/6
D2011  ; W50表示01行目  予備1   4/6
D2012  ; W50表示01行目  予備1   5/6
D2013  ; W50表示01行目  予備1   6/6
D2024  ; W50表示01行目  管径
D2025  ; W50表示01行目  肉厚
D2026  ; W50表示01行目  材質    1/4
D2027  ; W50表示01行目  材質    2/4
D2028  ; W50表示01行目  材質    3/4
D2029  ; W50表示01行目  材質    4/4
D2033  ; W50表示01行目  曲径1
D2034  ; W50表示01行目  曲径2
D2036  ; W50表示01行目  ﾜｰｸ全長
D2037  ; W50表示01行目  ﾜｰｸ全長
D2050  ; W50表示02行目  ﾊﾟｰﾂ№  1/8
D2051  ; W50表示02行目  ﾊﾟｰﾂ№  2/8
D2052  ; W50表示02行目  ﾊﾟｰﾂ№  3/8
D2053  ; W50表示02行目  ﾊﾟｰﾂ№  4/8
D2054  ; W50表示02行目  ﾊﾟｰﾂ№  5/8
D2055  ; W50表示02行目  ﾊﾟｰﾂ№  6/8
D2056  ; W50表示02行目  ﾊﾟｰﾂ№  7/8
D2057  ; W50表示02行目  ﾊﾟｰﾂ№  8/8
D2058  ; W50表示02行目  予備1   1/6
D2059  ; W50表示02行目  予備1   2/6
D2060  ; W50表示02行目  予備1   3/6
D2061  ; W50表示02行目  予備1   4/6
D2062  ; W50表示02行目  予備1   5/6
D2063  ; W50表示02行目  予備1   6/6
D2074  ; W50表示02行目  管径
D2075  ; W50表示02行目  肉厚
D2076  ; W50表示02行目  材質    1/4
D2077  ; W50表示02行目  材質    2/4
D2078  ; W50表示02行目  材質    3/4
D2079  ; W50表示02行目  材質    4/4
D2083  ; W50表示02行目  曲径1
D2084  ; W50表示02行目  曲径2
D2086  ; W50表示02行目  ﾜｰｸ全長
D2087  ; W50表示02行目  ﾜｰｸ全長
D2100  ; W50表示03行目  ﾊﾟｰﾂ№  1/8
D2101  ; W50表示03行目  ﾊﾟｰﾂ№  2/8
D2102  ; W50表示03行目  ﾊﾟｰﾂ№  3/8
D2103  ; W50表示03行目  ﾊﾟｰﾂ№  4/8
D2104  ; W50表示03行目  ﾊﾟｰﾂ№  5/8
D2105  ; W50表示03行目  ﾊﾟｰﾂ№  6/8
D2106  ; W50表示03行目  ﾊﾟｰﾂ№  7/8
D2107  ; W50表示03行目  ﾊﾟｰﾂ№  8/8
D2108  ; W50表示03行目  予備1   1/6
D2109  ; W50表示03行目  予備1   2/6
D2110  ; W50表示03行目  予備1   3/6
D2111  ; W50表示03行目  予備1   4/6
D2112  ; W50表示03行目  予備1   5/6
D2113  ; W50表示03行目  予備1   6/6
D2124  ; W50表示03行目  管径
D2125  ; W50表示03行目  肉厚
D2126  ; W50表示03行目  材質    1/4
D2127  ; W50表示03行目  材質    2/4
D2128  ; W50表示03行目  材質    3/4
D2129  ; W50表示03行目  材質    4/4
D2133  ; W50表示03行目  曲径1
D2134  ; W50表示03行目  曲径2
D2136  ; W50表示03行目  ﾜｰｸ全長
D2137  ; W50表示03行目  ﾜｰｸ全長
D2150  ; W50表示04行目  ﾊﾟｰﾂ№  1/8
D2151  ; W50表示04行目  ﾊﾟｰﾂ№  2/8
D2152  ; W50表示04行目  ﾊﾟｰﾂ№  3/8
D2153  ; W50表示04行目  ﾊﾟｰﾂ№  4/8
D2154  ; W50表示04行目  ﾊﾟｰﾂ№  5/8
D2155  ; W50表示04行目  ﾊﾟｰﾂ№  6/8
D2156  ; W50表示04行目  ﾊﾟｰﾂ№  7/8
D2157  ; W50表示04行目  ﾊﾟｰﾂ№  8/8
D2158  ; W50表示04行目  予備1   1/6
D2159  ; W50表示04行目  予備1   2/6
D2160  ; W50表示04行目  予備1   3/6
D2161  ; W50表示04行目  予備1   4/6
D2162  ; W50表示04行目  予備1   5/6
D2163  ; W50表示04行目  予備1   6/6
D2174  ; W50表示04行目  管径
D2175  ; W50表示04行目  肉厚
D2176  ; W50表示04行目  材質    1/4
D2177  ; W50表示04行目  材質    2/4
D2178  ; W50表示04行目  材質    3/4
D2179  ; W50表示04行目  材質    4/4
D2183  ; W50表示04行目  曲径1
D2184  ; W50表示04行目  曲径2
D2186  ; W50表示04行目  ﾜｰｸ全長
D2187  ; W50表示04行目  ﾜｰｸ全長
D2200  ; W50表示05行目  ﾊﾟｰﾂ№  1/8
D2201  ; W50表示05行目  ﾊﾟｰﾂ№  2/8
D2202  ; W50表示05行目  ﾊﾟｰﾂ№  3/8
D2203  ; W50表示05行目  ﾊﾟｰﾂ№  4/8
D2204  ; W50表示05行目  ﾊﾟｰﾂ№  5/8
D2205  ; W50表示05行目  ﾊﾟｰﾂ№  6/8
D2206  ; W50表示05行目  ﾊﾟｰﾂ№  7/8
D2207  ; W50表示05行目  ﾊﾟｰﾂ№  8/8
D2208  ; W50表示05行目  予備1   1/6
D2209  ; W50表示05行目  予備1   2/6
D2210  ; W50表示05行目  予備1   3/6
D2211  ; W50表示05行目  予備1   4/6
D2212  ; W50表示05行目  予備1   5/6
D2213  ; W50表示05行目  予備1   6/6
D2224  ; W50表示05行目  管径
D2225  ; W50表示05行目  肉厚
D2226  ; W50表示05行目  材質    1/4
D2227  ; W50表示05行目  材質    2/4
D2228  ; W50表示05行目  材質    3/4
D2229  ; W50表示05行目  材質    4/4
D2233  ; W50表示05行目  曲径1
D2234  ; W50表示05行目  曲径2
D2236  ; W50表示05行目  ﾜｰｸ全長
D2237  ; W50表示05行目  ﾜｰｸ全長
D2250  ; W50表示06行目  ﾊﾟｰﾂ№  1/8
D2251  ; W50表示06行目  ﾊﾟｰﾂ№  2/8
D2252  ; W50表示06行目  ﾊﾟｰﾂ№  3/8
D2253  ; W50表示06行目  ﾊﾟｰﾂ№  4/8
D2254  ; W50表示06行目  ﾊﾟｰﾂ№  5/8
D2255  ; W50表示06行目  ﾊﾟｰﾂ№  6/8
D2256  ; W50表示06行目  ﾊﾟｰﾂ№  7/8
D2257  ; W50表示06行目  ﾊﾟｰﾂ№  8/8
D2258  ; W50表示06行目  予備1   1/6
D2259  ; W50表示06行目  予備1   2/6
D2260  ; W50表示06行目  予備1   3/6
D2261  ; W50表示06行目  予備1   4/6
D2262  ; W50表示06行目  予備1   5/6
D2263  ; W50表示06行目  予備1   6/6
D2274  ; W50表示06行目  管径
D2275  ; W50表示06行目  肉厚
D2276  ; W50表示06行目  材質    1/4
D2277  ; W50表示06行目  材質    2/4
D2278  ; W50表示06行目  材質    3/4
D2279  ; W50表示06行目  材質    4/4
D2283  ; W50表示06行目  曲径1
D2284  ; W50表示06行目  曲径2
D2286  ; W50表示06行目  ﾜｰｸ全長
D2287  ; W50表示06行目  ﾜｰｸ全長
D2300  ; W50表示07行目  ﾊﾟｰﾂ№  1/8
D2301  ; W50表示07行目  ﾊﾟｰﾂ№  2/8
D2302  ; W50表示07行目  ﾊﾟｰﾂ№  3/8
D2303  ; W50表示07行目  ﾊﾟｰﾂ№  4/8
D2304  ; W50表示07行目  ﾊﾟｰﾂ№  5/8
D2305  ; W50表示07行目  ﾊﾟｰﾂ№  6/8
D2306  ; W50表示07行目  ﾊﾟｰﾂ№  7/8
D2307  ; W50表示07行目  ﾊﾟｰﾂ№  8/8
D2308  ; W50表示07行目  予備1   1/6
D2309  ; W50表示07行目  予備1   2/6
D2310  ; W50表示07行目  予備1   3/6
D2311  ; W50表示07行目  予備1   4/6
D2312  ; W50表示07行目  予備1   5/6
D2313  ; W50表示07行目  予備1   6/6
D2324  ; W50表示07行目  管径
D2325  ; W50表示07行目  肉厚
D2326  ; W50表示07行目  材質    1/4
D2327  ; W50表示07行目  材質    2/4
D2328  ; W50表示07行目  材質    3/4
D2329  ; W50表示07行目  材質    4/4
D2333  ; W50表示07行目  曲径1
D2334  ; W50表示07行目  曲径2
D2336  ; W50表示07行目  ﾜｰｸ全長
D2337  ; W50表示07行目  ﾜｰｸ全長
D2350  ; W50表示08行目  ﾊﾟｰﾂ№  1/8
D2351  ; W50表示08行目  ﾊﾟｰﾂ№  2/8
D2352  ; W50表示08行目  ﾊﾟｰﾂ№  3/8
D2353  ; W50表示08行目  ﾊﾟｰﾂ№  4/8
D2354  ; W50表示08行目  ﾊﾟｰﾂ№  5/8
D2355  ; W50表示08行目  ﾊﾟｰﾂ№  6/8
D2356  ; W50表示08行目  ﾊﾟｰﾂ№  7/8
D2357  ; W50表示08行目  ﾊﾟｰﾂ№  8/8
D2358  ; W50表示08行目  予備1   1/6
D2359  ; W50表示08行目  予備1   2/6
D2360  ; W50表示08行目  予備1   3/6
D2361  ; W50表示08行目  予備1   4/6
D2362  ; W50表示08行目  予備1   5/6
D2363  ; W50表示08行目  予備1   6/6
D2374  ; W50表示08行目  管径
D2375  ; W50表示08行目  肉厚
D2376  ; W50表示08行目  材質    1/4
D2377  ; W50表示08行目  材質    2/4
D2378  ; W50表示08行目  材質    3/4
D2379  ; W50表示08行目  材質    4/4
D2383  ; W50表示08行目  曲径1
D2384  ; W50表示08行目  曲径2
D2386  ; W50表示08行目  ﾜｰｸ全長
D2387  ; W50表示08行目  ﾜｰｸ全長
D2400  ; W50表示09行目  ﾊﾟｰﾂ№  1/8
D2401  ; W50表示09行目  ﾊﾟｰﾂ№  2/8
D2402  ; W50表示09行目  ﾊﾟｰﾂ№  3/8
D2403  ; W50表示09行目  ﾊﾟｰﾂ№  4/8
D2404  ; W50表示09行目  ﾊﾟｰﾂ№  5/8
D2405  ; W50表示09行目  ﾊﾟｰﾂ№  6/8
D2406  ; W50表示09行目  ﾊﾟｰﾂ№  7/8
D2407  ; W50表示09行目  ﾊﾟｰﾂ№  8/8
D2408  ; W50表示09行目  予備1   1/6
D2409  ; W50表示09行目  予備1   2/6
D2410  ; W50表示09行目  予備1   3/6
D2411  ; W50表示09行目  予備1   4/6
D2412  ; W50表示09行目  予備1   5/6
D2413  ; W50表示09行目  予備1   6/6
D2424  ; W50表示09行目  管径
D2425  ; W50表示09行目  肉厚
D2426  ; W50表示09行目  材質    1/4
D2427  ; W50表示09行目  材質    2/4
D2428  ; W50表示09行目  材質    3/4
D2429  ; W50表示09行目  材質    4/4
D2433  ; W50表示09行目  曲径1
D2434  ; W50表示09行目  曲径2
D2436  ; W50表示09行目  ﾜｰｸ全長
D2437  ; W50表示09行目  ﾜｰｸ全長
D2450  ; W50表示10行目  ﾊﾟｰﾂ№  1/8
D2451  ; W50表示10行目  ﾊﾟｰﾂ№  2/8
D2452  ; W50表示10行目  ﾊﾟｰﾂ№  3/8
D2453  ; W50表示10行目  ﾊﾟｰﾂ№  4/8
D2454  ; W50表示10行目  ﾊﾟｰﾂ№  5/8
D2455  ; W50表示10行目  ﾊﾟｰﾂ№  6/8
D2456  ; W50表示10行目  ﾊﾟｰﾂ№  7/8
D2457  ; W50表示10行目  ﾊﾟｰﾂ№  8/8
D2458  ; W50表示10行目  予備1   1/6
D2459  ; W50表示10行目  予備1   2/6
D2460  ; W50表示10行目  予備1   3/6
D2461  ; W50表示10行目  予備1   4/6
D2462  ; W50表示10行目  予備1   5/6
D2463  ; W50表示10行目  予備1   6/6
D2474  ; W50表示10行目  管径
D2475  ; W50表示10行目  肉厚
D2476  ; W50表示10行目  材質    1/4
D2477  ; W50表示10行目  材質    2/4
D2478  ; W50表示10行目  材質    3/4
D2479  ; W50表示10行目  材質    4/4
D2483  ; W50表示10行目  曲径1
D2484  ; W50表示10行目  曲径2
D2486  ; W50表示10行目  ﾜｰｸ全長
D2487  ; W50表示10行目  ﾜｰｸ全長
D3001  ; 前ｽｷｬﾝ異常2
D3003  ; 前ｽｷｬﾝ異常4
D3011  ; 新異常2
D3013  ; 新異常4
D3020  ; ｽﾘｰﾌﾞ長さPT開始時記憶
D3021  ; ｸﾗﾝﾌﾟ長さC開始時記憶
D3023  ; ﾌﾟﾚｯｼｬ長さPL開始時記憶
D3024  ; 管径開始時記憶
D3025  ; 肉厚開始時記憶
D3026  ; 材質開始時記憶
D3030  ; ﾜｰｸﾃﾞｰﾀ ｽﾘｰﾌﾞ開始時記憶
D3033  ; 曲げ半径開始時記憶
D3100  ; tan(CM0/2)/*R
D3101  ; tan(CM0/2)/*R
D3102  ; tan(CM1/2)/*R
D3103  ; tan(CM1/2)/*R
D3122  ; tan(CM11/2)/*R
D3123  ; tan(CM11/2)/*R
D3127  ; 曲げ径FLT
D3131  ; C0-CM0/2*2π*R/360
D3133  ; C1-CM1/2*2π*R/360
D3157  ; 2π*R/360
D3161  ; 曲げ周長の合計
D3163  ; Yの合計
D3171  ; 固定SB_DW
D3173  ; 比例SB_DW
D3201  ; 比例SB‗FLT
D3203  ; 比例SB‗FLT/100
D3207  ; 1-比例SB/100‗FLT
D3209  ; Cn‗FLT
D3213  ; Cn/(1-比例SB)‗FLT
D3215  ; Cn/(1-比例SB)‗INT
D3251  ; 比例SB‗FLT
D3253  ; 比例SB‗FLT/100
D3257  ; 1+比例SB/100‗FLT
D3259  ; Cn‗FLT
D3263  ; Cn/(1-比例SB)‗FLT
D3265  ; Cn/(1-比例SB)‗INT
D5803  ; 1回転あたりのﾊﾟﾙｽ_2W
D5805  ; 1回転あたりの移動量_2W
D5806  ; 始動時ﾊﾞｲｱｽ速度_2W
D5807  ; 始動時ﾊﾞｲｱｽ速度_2W
D5826  ; ﾄﾙｸ制限値
D5873  ; 原点ｱﾄﾞﾚｽ
D5886  ; 原点復帰トルク制限値
D5888  ; 加速時間変更値
D5889  ; 加速時間変更値
D5890  ; 減速時間変更値
D5891  ; 減速時間変更値
D5892  ; 加減速変更許可
D5901  ; Pr.101
D5904  ; Pr.104機能選択A-1
D5905  ; Pr.105
D5906  ; Pr.106
D5907  ; Pr.107
D5911  ; Pr.111
D5912  ; Pr.112
D5913  ; Pr.113
D5916  ; Pr.116
D5917  ; Pr.117
D5918  ; Pr.118
D5919  ; Pr.119
D5920  ; Pr.120
D6000  ; D60=001 ｸﾗﾝﾌﾟ閉
D6001  ; D61=001 ﾌﾟﾚｯｼｬ閉
D6002  ; D60=005 ﾁｬｯｸ開
D6003  ; D61=005 ﾌﾗﾝｼﾞ穴検上昇
D6005  ; D60=012 送り原点復帰指令
D6008  ; D60=040 ﾋﾈﾘ原点復帰指令
D6009  ; D61=041 芯金後退
D6010  ; D62=040 曲げ戻り
D6013  ; D60=055 ｷｬﾚｯｼﾞ横移動R小
D6014  ; D61=055 芯金横移動R小
D6017  ; D60=070 送りYLD位置
D6019  ; D60=999 原点復帰完了
D6820  ; [TP]W050角度値  入力
D6822  ; SB      算出角度
D7022  ; ﾊﾟｲﾌﾟ径***A～***A
D7023  ; 管外形***A～***A
D7024  ; 管外形200A～予備1
D7025  ; 管外形予備1～予備2
D7720  ; 曲げ    減速角度
D7721  ; 曲げ    減速角度
R61  ; 始点金物_ＤＣ
R62  ; 始点金物_ＦＥ
R63  ; 始点金物_ＨＧ
R65  ; ﾌﾗﾝｼﾞ圧力
R67  ; 終点金物_ＨＧ
R80  ; ｻｲﾄﾞﾌﾞｰｽﾀｰ圧力_***%
R82  ; ﾌﾟﾚｯｼｬｰ圧力_***%
R84  ; ﾊﾞｯｸﾌﾞｰｽﾀﾃｰﾌﾞﾙ_*
R86  ; ｸﾗﾝﾌﾟ長_****.*mm
R88  ; ﾌﾟﾚｯｼｬｰ長_****.*mm
R101  ; BT_2
R102  ; BT_3
R103  ; BT_4
R104  ; BT_5
R105  ; BT_6
R106  ; BT_7
R107  ; BT_8
R108  ; BT_9
R109  ; BT_10
R110  ; BT_11
R111  ; BT_12
R112  ; BT_13
R113  ; BT_14
R114  ; BT_15
R115  ; BT_16
R116  ; BT_17
R117  ; BT_18
R118  ; BT_19
R119  ; BT_20
R120  ; BT_21
R121  ; BT_22
R122  ; BT_23
R123  ; BT_24
R124  ; BT_25
R125  ; BT_26
R126  ; BT_27
R127  ; BT_28
R128  ; BT_29
R129  ; BT_30
R302  ; Y軸ﾏｽﾀｰ曲げ 2段
R304  ; Y軸ﾏｽﾀｰ曲げ 3段
R306  ; Y軸ﾏｽﾀｰ曲げ 4段
R308  ; Y軸ﾏｽﾀｰ曲げ 5段
R310  ; Y軸ﾏｽﾀｰ曲げ 6段
R312  ; Y軸ﾏｽﾀｰ曲げ 7段
R314  ; Y軸ﾏｽﾀｰ曲げ 8段
R316  ; Y軸ﾏｽﾀｰ曲げ 9段
R318  ; Y軸ﾏｽﾀｰ曲げ10段
R320  ; Y軸ﾏｽﾀｰ曲げ11段
R322  ; Y軸ﾏｽﾀｰ曲げ12段
R324  ; Y軸ﾏｽﾀｰ曲げ13段
R326  ; Y軸ﾏｽﾀｰ曲げ14段
R328  ; Y軸ﾏｽﾀｰ曲げ15段
R330  ; Y軸ﾏｽﾀｰ曲げ16段
R332  ; Y軸ﾏｽﾀｰ曲げ17段
R334  ; Y軸ﾏｽﾀｰ曲げ18段
R336  ; Y軸ﾏｽﾀｰ曲げ19段
R338  ; Y軸ﾏｽﾀｰ曲げ20段
R340  ; Y軸ﾏｽﾀｰ曲げ21段
R342  ; Y軸ﾏｽﾀｰ曲げ22段
R344  ; Y軸ﾏｽﾀｰ曲げ23段
R346  ; Y軸ﾏｽﾀｰ曲げ24段
R348  ; Y軸ﾏｽﾀｰ曲げ25段
R350  ; Y軸ﾏｽﾀｰ曲げ26段
R352  ; Y軸ﾏｽﾀｰ曲げ27段
R354  ; Y軸ﾏｽﾀｰ曲げ28段
R356  ; Y軸ﾏｽﾀｰ曲げ29段
R358  ; Y軸ﾏｽﾀｰ曲げ30段
R372  ; B軸ﾏｽﾀｰ曲げ 2段
R374  ; B軸ﾏｽﾀｰ曲げ 3段
R376  ; B軸ﾏｽﾀｰ曲げ 4段
R378  ; B軸ﾏｽﾀｰ曲げ 5段
R380  ; B軸ﾏｽﾀｰ曲げ 6段
R382  ; B軸ﾏｽﾀｰ曲げ 7段
R384  ; B軸ﾏｽﾀｰ曲げ 8段
R386  ; B軸ﾏｽﾀｰ曲げ 9段
R388  ; B軸ﾏｽﾀｰ曲げ 10段
R390  ; B軸ﾏｽﾀｰ曲げ 11段
R392  ; B軸ﾏｽﾀｰ曲げ 12段
R394  ; B軸ﾏｽﾀｰ曲げ 13段
R396  ; B軸ﾏｽﾀｰ曲げ 14段
R398  ; B軸ﾏｽﾀｰ曲げ 15段
R400  ; B軸ﾏｽﾀｰ曲げ 16段
R402  ; B軸ﾏｽﾀｰ曲げ 17段
R404  ; B軸ﾏｽﾀｰ曲げ 18段
R406  ; B軸ﾏｽﾀｰ曲げ 19段
R408  ; B軸ﾏｽﾀｰ曲げ 20段
R410  ; B軸ﾏｽﾀｰ曲げ 21段
R412  ; B軸ﾏｽﾀｰ曲げ 22段
R414  ; B軸ﾏｽﾀｰ曲げ 23段
R416  ; B軸ﾏｽﾀｰ曲げ 24段
R418  ; B軸ﾏｽﾀｰ曲げ 25段
R420  ; B軸ﾏｽﾀｰ曲げ 26段
R422  ; B軸ﾏｽﾀｰ曲げ 27段
R424  ; B軸ﾏｽﾀｰ曲げ 28段
R426  ; B軸ﾏｽﾀｰ曲げ 29段
R428  ; B軸ﾏｽﾀｰ曲げ 30段
R442  ; C軸ﾏｽﾀｰ曲げ 2段
R444  ; C軸ﾏｽﾀｰ曲げ 3段
R446  ; C軸ﾏｽﾀｰ曲げ 4段
R448  ; C軸ﾏｽﾀｰ曲げ 5段
R450  ; C軸ﾏｽﾀｰ曲げ 6段
R452  ; C軸ﾏｽﾀｰ曲げ 7段
R454  ; C軸ﾏｽﾀｰ曲げ 8段
R456  ; C軸ﾏｽﾀｰ曲げ 9段
R458  ; C軸ﾏｽﾀｰ曲げ10段
R460  ; C軸ﾏｽﾀｰ曲げ11段
R462  ; C軸ﾏｽﾀｰ曲げ12段
R464  ; C軸ﾏｽﾀｰ曲げ13段
R466  ; C軸ﾏｽﾀｰ曲げ14段
R468  ; C軸ﾏｽﾀｰ曲げ15段
R470  ; C軸ﾏｽﾀｰ曲げ16段
R472  ; C軸ﾏｽﾀｰ曲げ17段
R474  ; C軸ﾏｽﾀｰ曲げ18段
R476  ; C軸ﾏｽﾀｰ曲げ19段
R478  ; C軸ﾏｽﾀｰ曲げ20段
R480  ; C軸ﾏｽﾀｰ曲げ21段
R482  ; C軸ﾏｽﾀｰ曲げ22段
R484  ; C軸ﾏｽﾀｰ曲げ23段
R486  ; C軸ﾏｽﾀｰ曲げ24段
R488  ; C軸ﾏｽﾀｰ曲げ25段
R490  ; C軸ﾏｽﾀｰ曲げ26段
R492  ; C軸ﾏｽﾀｰ曲げ27段
R494  ; C軸ﾏｽﾀｰ曲げ28段
R496  ; C軸ﾏｽﾀｰ曲げ29段
R498  ; C軸ﾏｽﾀｰ曲げ30段
R617  ; Y軸曲げﾃﾞｰﾀ 2段
R619  ; Y軸曲げﾃﾞｰﾀ 3段
R621  ; Y軸曲げﾃﾞｰﾀ 4段
R623  ; Y軸曲げﾃﾞｰﾀ 5段
R625  ; Y軸曲げﾃﾞｰﾀ 6段
R627  ; Y軸曲げﾃﾞｰﾀ 7段
R629  ; Y軸曲げﾃﾞｰﾀ 8段
R631  ; Y軸曲げﾃﾞｰﾀ 9段
R633  ; Y軸曲げﾃﾞｰﾀ 10段
R635  ; Y軸曲げﾃﾞｰﾀ 11段
R637  ; Y軸曲げﾃﾞｰﾀ 12段
R639  ; Y軸曲げﾃﾞｰﾀ 13段
R641  ; Y軸曲げﾃﾞｰﾀ 14段
R643  ; Y軸曲げﾃﾞｰﾀ 15段
R645  ; Y軸曲げﾃﾞｰﾀ 16段
R647  ; Y軸曲げﾃﾞｰﾀ 17段
R649  ; Y軸曲げﾃﾞｰﾀ 18段
R651  ; Y軸曲げﾃﾞｰﾀ 19段
R653  ; Y軸曲げﾃﾞｰﾀ 20段
R655  ; Y軸曲げﾃﾞｰﾀ 21段
R657  ; Y軸曲げﾃﾞｰﾀ 22段
R659  ; Y軸曲げﾃﾞｰﾀ 23段
R661  ; Y軸曲げﾃﾞｰﾀ 24段
R663  ; Y軸曲げﾃﾞｰﾀ 25段
R665  ; Y軸曲げﾃﾞｰﾀ 26段
R667  ; Y軸曲げﾃﾞｰﾀ 27段
R669  ; Y軸曲げﾃﾞｰﾀ 28段
R671  ; Y軸曲げﾃﾞｰﾀ 29段
R673  ; Y軸曲げﾃﾞｰﾀ 30段
R695  ; B軸ﾜｰｸ曲げ 6段
R697  ; B軸ﾜｰｸ曲げ 7段
R699  ; B軸ﾜｰｸ曲げ 8段
R701  ; B軸ﾜｰｸ曲げ 9段
R703  ; B軸ﾜｰｸ曲げ 10段
R705  ; B軸ﾜｰｸ曲げ 11段
R707  ; B軸ﾜｰｸ曲げ 12段
R709  ; B軸ﾜｰｸ曲げ 13段
R711  ; B軸ﾜｰｸ曲げ 14段
R713  ; B軸ﾜｰｸ曲げ 15段
R715  ; B軸ﾜｰｸ曲げ 16段
R717  ; B軸ﾜｰｸ曲げ 17段
R719  ; B軸ﾜｰｸ曲げ 18段
R721  ; B軸ﾜｰｸ曲げ 19段
R723  ; B軸ﾜｰｸ曲げ 20段
R725  ; B軸ﾜｰｸ曲げ 21段
R727  ; B軸ﾜｰｸ曲げ 22段
R729  ; B軸ﾜｰｸ曲げ 23段
R731  ; B軸ﾜｰｸ曲げ 24段
R733  ; B軸ﾜｰｸ曲げ 25段
R735  ; B軸ﾜｰｸ曲げ 26段
R737  ; B軸ﾜｰｸ曲げ 27段
R739  ; B軸ﾜｰｸ曲げ 28段
R741  ; B軸ﾜｰｸ曲げ 29段
R743  ; B軸ﾜｰｸ曲げ 30段
R757  ; C軸ﾜｰｸ曲げ 2段
R759  ; C軸ﾜｰｸ曲げ 3段
R761  ; C軸ﾜｰｸ曲げ 4段
R763  ; C軸ﾜｰｸ曲げ 5段
R765  ; C軸ﾜｰｸ曲げ 6段
R767  ; C軸ﾜｰｸ曲げ 7段
R769  ; C軸ﾜｰｸ曲げ 8段
R771  ; C軸ﾜｰｸ曲げ 9段
R773  ; C軸ﾜｰｸ曲げ10段
R775  ; C軸ﾜｰｸ曲げ11段
R777  ; C軸ﾜｰｸ曲げ12段
R779  ; C軸ﾜｰｸ曲げ13段
R781  ; C軸ﾜｰｸ曲げ14段
R783  ; C軸ﾜｰｸ曲げ15段
R785  ; C軸ﾜｰｸ曲げ16段
R787  ; C軸ﾜｰｸ曲げ17段
R789  ; C軸ﾜｰｸ曲げ18段
R791  ; C軸ﾜｰｸ曲げ19段
R793  ; C軸ﾜｰｸ曲げ20段
R795  ; C軸ﾜｰｸ曲げ21段
R797  ; C軸ﾜｰｸ曲げ22段
R799  ; C軸ﾜｰｸ曲げ23段
R801  ; C軸ﾜｰｸ曲げ24段
R803  ; C軸ﾜｰｸ曲げ25段
R805  ; C軸ﾜｰｸ曲げ26段
R807  ; C軸ﾜｰｸ曲げ27段
R809  ; C軸ﾜｰｸ曲げ28段
R811  ; C軸ﾜｰｸ曲げ29段
R813  ; C軸ﾜｰｸ曲げ30段
R1100  ; ﾘﾓｰﾄﾜｰｸ選択No.
R3000  ; S管 65A SGP 比例SB
R3001  ; S管 65A #40 比例SB
R3002  ; S管 65A #80 比例SB
R3010  ; S管 65A SGP 固定SB
R3011  ; S管 65A #40 固定SB
R3012  ; S管 65A #80 固定SB
R3020  ; S管 80A SGP 比例SB
R3021  ; S管 80A #40 比例SB
R3022  ; S管 80A #80 比例SB
R3030  ; S管 80A SGP 固定SB
R3031  ; S管 80A #40 固定SB
R3032  ; S管 80A #80 固定SB
R3040  ; S管 100A SGP 比例SB
R3041  ; S管 100A #40 比例SB
R3042  ; S管 100A #80 比例SB
R3050  ; S管 100A SGP 固定SB
R3051  ; S管 100A #40 固定SB
R3052  ; S管 100A #80 固定SB
R3060  ; S管 200A SGP 比例SB
R3061  ; S管 200A #40 比例SB
R3062  ; S管 200A #80 比例SB
R3070  ; S管 200A SGP 固定SB
R3071  ; S管 200A #40 固定SB
R3072  ; S管 200A #80 固定SB
R3100  ; E管 65A SGP 比例SB
R3101  ; E管 65A #40 比例SB
R3102  ; E管 65A #80 比例SB
R3110  ; E管 65A SGP 固定SB
R3111  ; E管 65A #40 固定SB
R3112  ; E管 65A #80 固定SB
R3120  ; E管 80A SGP 比例SB
R3121  ; E管 80A #40 比例SB
R3122  ; E管 80A #80 比例SB
R3130  ; E管 80A SGP 固定SB
R3131  ; E管 80A #40 固定SB
R3132  ; E管 80A #80 固定SB
R3140  ; E管 100A SGP 比例SB
R3141  ; E管 100A #40 比例SB
R3142  ; E管 100A #80 比例SB
R3150  ; E管 100A SGP 固定SB
R3151  ; E管 100A #40 固定SB
R3152  ; E管 100A #80 固定SB
R3160  ; E管 200A SGP 比例SB
R3161  ; E管 200A #40 比例SB
R3162  ; E管 200A #80 比例SB
R3170  ; E管 200A SGP 固定SB
R3171  ; E管 200A #40 固定SB
R3172  ; E管 200A #80 固定SB
R3300  ; S管 65A SGPﾌﾟﾚｯｼｬ圧力
R3301  ; S管 65A #40ﾌﾟﾚｯｼｬ圧力
R3302  ; S管 65A #80ﾌﾟﾚｯｼｬ圧力
R3310  ; S管 65A SGPｻｲﾄﾞﾌﾞｰｽﾀ圧力
R3311  ; S管 65A #40ｻｲﾄﾞﾌﾞｰｽﾀ圧力
R3312  ; S管 65A #80ｻｲﾄﾞﾌﾞｰｽﾀ圧力
R3320  ; S管 80A SGPﾌﾟﾚｯｼｬ圧力
R3321  ; S管 80A #40ﾌﾟﾚｯｼｬ圧力
R3322  ; S管 80A #80ﾌﾟﾚｯｼｬ圧力
R3330  ; S管 80A SGPｻｲﾄﾞﾌﾞｰｽﾀ圧力
R3331  ; S管 80A #40ｻｲﾄﾞﾌﾞｰｽﾀ圧力
R3332  ; S管 80A #80ｻｲﾄﾞﾌﾞｰｽﾀ圧力
R3340  ; S管 100A SGPﾌﾟﾚｯｼｬ圧力
R3341  ; S管 100A #40ﾌﾟﾚｯｼｬ圧力
R3342  ; S管 100A #80ﾌﾟﾚｯｼｬ圧力
R3350  ; S管 100A SGPｻｲﾄﾞﾌﾞｰｽﾀ圧力
R3351  ; S管 100A #40ｻｲﾄﾞﾌﾞｰｽﾀ圧力
R3352  ; S管 100A #80ｻｲﾄﾞﾌﾞｰｽﾀ圧力
R3360  ; S管 200A SGP
R3361  ; S管 200A #40
R3362  ; S管 200A #80
R3370  ; S管 200A SGP
R3371  ; S管 200A #40
R3372  ; S管 200A #80
R3400  ; E管 65A SGPﾌﾟﾚｯｼｬ圧力
R3401  ; E管 65A #40ﾌﾟﾚｯｼｬ圧力
R3402  ; E管 65A #80ﾌﾟﾚｯｼｬ圧力
R3410  ; E管 65A SGPｻｲﾄﾞﾌﾞｰｽﾀ圧力
R3411  ; E管 65A #40ｻｲﾄﾞﾌﾞｰｽﾀ圧力
R3412  ; E管 65A #80ｻｲﾄﾞﾌﾞｰｽﾀ圧力
R3420  ; E管 80A SGPﾌﾟﾚｯｼｬ圧力
R3421  ; E管 80A #40ﾌﾟﾚｯｼｬ圧力
R3422  ; E管 80A #80ﾌﾟﾚｯｼｬ圧力
R3430  ; E管 80A SGPｻｲﾄﾞﾌﾞｰｽﾀ圧力
R3431  ; E管 80A #40ｻｲﾄﾞﾌﾞｰｽﾀ圧力
R3432  ; E管 80A #80ｻｲﾄﾞﾌﾞｰｽﾀ圧力
R3440  ; E管 100A SGPﾌﾟﾚｯｼｬ圧力
R3441  ; E管 100A #40ﾌﾟﾚｯｼｬ圧力
R3442  ; E管 100A #80ﾌﾟﾚｯｼｬ圧力
R3450  ; E管 100A SGPｻｲﾄﾞﾌﾞｰｽﾀ圧力
R3451  ; E管 100A #40ｻｲﾄﾞﾌﾞｰｽﾀ圧力
R3452  ; E管 100A #80ｻｲﾄﾞﾌﾞｰｽﾀ圧力
R3460  ; E管 200A SGP
R3461  ; E管 200A #40
R3462  ; E管 200A #80
R3470  ; E管 200A SGP
R3471  ; E管 200A #40
R3472  ; E管 200A #80
R20006  ; W50_ST先頭
R20007  ; W50_STｶｰｿﾙ表示
R20009  ; W50_STｶｰｿﾙ1ｽｷｬﾝ遅延
R20017  ; ﾃﾞｰﾀ異常
R20018  ; ﾃﾞｰﾀ異常番号
R20023  ; 送りﾌﾗﾝｼﾞ待機+α
R20025  ; ﾁｬｯｸ上昇待機位置
R20026  ; 送りｽﾘｰﾌﾞ待機+α
R20027  ; 送りｽﾘｰﾌﾞ待機+α
R20030  ; 次段管径
R20031  ; 次段ﾌﾗﾝｼﾞ圧力
R20033  ; 次段送りﾌﾗﾝｼﾞ待機+α
R20035  ; 次段ﾁｬｯｸ上昇待機位置
R20036  ; 次段待機+α
R20037  ; 次段待機+α
R20071  ; 2段ﾃﾞｰﾀ異常番号
R20072  ; 3段ﾃﾞｰﾀ異常番号
R20073  ; 4段ﾃﾞｰﾀ異常番号
R20074  ; 5段ﾃﾞｰﾀ異常番号
R20075  ; 6段ﾃﾞｰﾀ異常番号
R20076  ; 7段ﾃﾞｰﾀ異常番号
R20077  ; 8段ﾃﾞｰﾀ異常番号
R20078  ; 9段ﾃﾞｰﾀ異常番号
R20079  ; 10段ﾃﾞｰﾀ異常番号
R20080  ; 11段ﾃﾞｰﾀ異常番号
R20081  ; 12段ﾃﾞｰﾀ異常番号
R20082  ; 13段ﾃﾞｰﾀ異常番号
R20083  ; 14段ﾃﾞｰﾀ異常番号
R20084  ; 15段ﾃﾞｰﾀ異常番号
R20085  ; 16段ﾃﾞｰﾀ異常番号
R20086  ; 17段ﾃﾞｰﾀ異常番号
R20087  ; 18段ﾃﾞｰﾀ異常番号
R20088  ; 19段ﾃﾞｰﾀ異常番号
R20089  ; 20段ﾃﾞｰﾀ異常番号
R20090  ; 21段ﾃﾞｰﾀ異常番号
R20091  ; 22段ﾃﾞｰﾀ異常番号
R20092  ; 23段ﾃﾞｰﾀ異常番号
R20093  ; 24段ﾃﾞｰﾀ異常番号
R20094  ; 25段ﾃﾞｰﾀ異常番号
R20095  ; 26段ﾃﾞｰﾀ異常番号
R20096  ; 27段ﾃﾞｰﾀ異常番号
R20097  ; 28段ﾃﾞｰﾀ異常番号
R20098  ; 29段ﾃﾞｰﾀ異常番号
R20099  ; 30段ﾃﾞｰﾀ異常番号
R20120  ; 送り低速速度
R20122  ; 送り端面検出速度
R20142  ; 送り原点許容範囲
R20156  ; 送りﾁｬｯｸ開位置
R20168  ; 送りﾊﾟｲﾌﾟ受け下降位置
R20194  ; 送りｽﾘｰﾌﾞ
R20204  ; 捻り_自動速度設定_TI
R20206  ; 捻り_手動速度設定_TI
R20208  ; 捻り_原点復帰速度設定_TI
R20240  ; 捻り_動作圧力
R20256  ; 捻り_B軸終ﾌﾘ_Work
R20306  ; 曲げ手動高速速度設定_TI
R20366  ; 曲げ曲げ戻り動作圧力
R20488  ; ﾍｯﾄﾞｼﾌﾄR大減速開始領域
R20490  ; ﾍｯﾄﾞｼﾌﾄR小減速開始領域
R20600  ; ｻｲﾄﾞﾌﾞｰｽﾀ65A_速度設定値
R20602  ; ｻｲﾄﾞﾌﾞｰｽﾀ80A_速度設定値
R20604  ; ｻｲﾄﾞﾌﾞｰｽﾀ100A_速度設定値
R20622  ; ｻｲﾄﾞﾌﾞｰｽﾀｼﾘﾝﾀﾞｽﾄﾛｰｸ
R20682  ; ﾁｬｯｸ最大設定値 (*3)
R20710  ; ﾁｬｯｸ上昇端(送り65A前端前)
R20712  ; ﾁｬｯｸ上昇端(送り65A前端後)
R20714  ; ﾁｬｯｸｽﾘｰﾌﾞ有時待機+α
R20716  ; ﾁｬｯｸｽﾘｰﾌﾞ有時待機+α
R20730  ; ﾁｬｯｸ送り現在値による前進端
R20752  ; 芯金前進側動作圧力
R20754  ; 芯金後退側動作圧力
R20756  ; ﾁｬｯｸ閉側低圧動作圧力
R20758  ; ﾁｬｯｸ閉側高圧動作圧力
R20760  ; ｵﾝﾛｰﾄﾞ動作圧力
R20762  ; ｳｫｰﾐﾝｸﾞｱｯﾌﾟ圧力
R20770  ; ﾌﾟﾚｯｼｬ動作圧力
R20800  ; PV2_ｵﾝﾛｰﾄﾞ強制1範囲
R20801  ; PV2_ｵﾝﾛｰﾄﾞ強制2範囲
R20802  ; PV2_ｵﾝﾛｰﾄﾞ強制3範囲
R20803  ; PV2_ｵﾝﾛｰﾄﾞ強制4範囲
R20804  ; PV2_強制設定値
R20805  ; PV2_最大設定比率
R20807  ; PV2_NULL
R20808  ; PV2_GAIN
R20810  ; PV2_ｵﾝﾛｰﾄﾞ強制1a
R20811  ; PV2_ｵﾝﾛｰﾄﾞ強制2a
R20812  ; PV2_ｵﾝﾛｰﾄﾞ強制3a
R20813  ; PV2_ｵﾝﾛｰﾄﾞ強制4a
R20814  ; PV2_ｵﾝﾛｰﾄﾞ強制5a
R20815  ; PV2_ｵﾝﾛｰﾄﾞ強制1b
R20816  ; PV2_ｵﾝﾛｰﾄﾞ強制2b
R20817  ; PV2_ｵﾝﾛｰﾄﾞ強制3b
R20818  ; PV2_ｵﾝﾛｰﾄﾞ強制4b
R20819  ; PV2_ｵﾝﾛｰﾄﾞ強制5b
R20830  ; PV3_ｵﾝﾛｰﾄﾞ強制1範囲
R20831  ; PV3_ｵﾝﾛｰﾄﾞ強制2範囲
R20832  ; PV3_ｵﾝﾛｰﾄﾞ強制3範囲
R20833  ; PV3_ｵﾝﾛｰﾄﾞ強制4範囲
R20834  ; PV3_強制設定値
R20835  ; PV3_最大設定比率
R20837  ; PV3_NULL
R20838  ; PV3_GAIN
R20840  ; PV3_ｵﾝﾛｰﾄﾞ強制1a
R20841  ; PV3_ｵﾝﾛｰﾄﾞ強制2a
R20842  ; PV3_ｵﾝﾛｰﾄﾞ強制3a
R20843  ; PV3_ｵﾝﾛｰﾄﾞ強制4a
R20844  ; PV3_ｵﾝﾛｰﾄﾞ強制5a
R20845  ; PV3_ｵﾝﾛｰﾄﾞ強制1b
R20846  ; PV3_ｵﾝﾛｰﾄﾞ強制2b
R20847  ; PV3_ｵﾝﾛｰﾄﾞ強制3b
R20848  ; PV3_ｵﾝﾛｰﾄﾞ強制4b
R20849  ; PV3_ｵﾝﾛｰﾄﾞ強制5b
R20860  ; PV4_ｵﾝﾛｰﾄﾞ強制1範囲
R20861  ; PV4_ｵﾝﾛｰﾄﾞ強制2範囲
R20862  ; PV4_ｵﾝﾛｰﾄﾞ強制3範囲
R20863  ; PV4_ｵﾝﾛｰﾄﾞ強制4範囲
R20864  ; PV4_強制設定値
R20865  ; PV4_最大設定比率
R20867  ; PV4_NULL
R20868  ; PV4_GAIN
R20870  ; PV4_ｵﾝﾛｰﾄﾞ強制1a
R20871  ; PV4_ｵﾝﾛｰﾄﾞ強制2a
R20872  ; PV4_ｵﾝﾛｰﾄﾞ強制3a
R20873  ; PV4_ｵﾝﾛｰﾄﾞ強制4a
R20874  ; PV4_ｵﾝﾛｰﾄﾞ強制5a
R20875  ; PV4_ｵﾝﾛｰﾄﾞ強制1b
R20876  ; PV4_ｵﾝﾛｰﾄﾞ強制2b
R20877  ; PV4_ｵﾝﾛｰﾄﾞ強制3b
R20878  ; PV4_ｵﾝﾛｰﾄﾞ強制4b
R20879  ; PV4_ｵﾝﾛｰﾄﾞ強制5b
R20940  ; 100%出力時
R20952  ; PV2油圧制御値_X3#.#Mpa
R20953  ; PV2油圧制御値_X4#.#Mpa
R20954  ; PV2油圧制御値_X5#.#Mpa
R20955  ; PV2油圧制御値_X6#.#Mpa
R20956  ; PV2油圧制御値_X7#.#Mpa
R20957  ; PV2油圧制御値_X8#.#Mpa
R20958  ; PV2油圧制御値_X9#.#Mpa
R20962  ; PV2油圧測定値_Y3#.#Mpa
R20963  ; PV2油圧測定値_Y4#.#Mpa
R20964  ; PV2油圧測定値_Y5#.#Mpa
R20965  ; PV2油圧測定値_Y6#.#Mpa
R20966  ; PV2油圧測定値_Y7#.#Mpa
R20967  ; PV2油圧測定値_Y8#.#Mpa
R20968  ; PV2油圧測定値_Y9#.#Mpa
R20972  ; PV3油圧制御値_X3#.#Mpa
R20973  ; PV3油圧制御値_X4#.#Mpa
R20974  ; PV3油圧制御値_X5#.#Mpa
R20975  ; PV3油圧制御値_X6#.#Mpa
R20976  ; PV3油圧制御値_X7#.#Mpa
R20977  ; PV3油圧制御値_X8#.#Mpa
R20978  ; PV3油圧制御値_X9#.#Mpa
R20982  ; PV3油圧測定値_Y3#.#Mpa
R20983  ; PV3油圧測定値_Y4#.#Mpa
R20984  ; PV3油圧測定値_Y5#.#Mpa
R20985  ; PV3油圧測定値_Y6#.#Mpa
R20986  ; PV3油圧測定値_Y7#.#Mpa
R20987  ; PV3油圧測定値_Y8#.#Mpa
R20988  ; PV3油圧測定値_Y9#.#Mpa
R20992  ; PV4油圧制御値_X3#.#Mpa
R20993  ; PV4油圧制御値_X4#.#Mpa
R20994  ; PV4油圧制御値_X5#.#Mpa
R20995  ; PV4油圧制御値_X6#.#Mpa
R20996  ; PV4油圧制御値_X7#.#Mpa
R20997  ; PV4油圧制御値_X8#.#Mpa
R20998  ; PV4油圧制御値_X9#.#Mpa
R21002  ; PV4油圧測定値_Y3#.#Mpa
R21003  ; PV4油圧測定値_Y4#.#Mpa
R21004  ; PV4油圧測定値_Y5#.#Mpa
R21005  ; PV4油圧測定値_Y6#.#Mpa
R21006  ; PV4油圧測定値_Y7#.#Mpa
R21007  ; PV4油圧測定値_Y8#.#Mpa
R21008  ; PV4油圧測定値_Y9#.#Mpa
R21108  ; ﾊﾟｲﾌﾟ計算長####.#mm
R21109  ; ﾊﾟｲﾌﾟ計算長####.#mm
R21110  ; ﾊﾟｲﾌﾟ最終段後余長####.#mm
R22086  ; 曲げ圧抜き確認
R22092  ; ｸﾗﾝﾌﾟﾀﾞｲ前進端遅延
R22093  ; ｸﾗﾝﾌﾟﾀﾞｲ後退端遅延
R22102  ; ﾌﾟﾚｯｼｬﾀﾞｲ前進端遅延
R22103  ; ﾌﾟﾚｯｼｬﾀﾞｲ後退端遅延
R22144  ; ﾁｬｯｸｴﾝｺｰﾀﾞ異常検出時間
R22156  ; 芯金圧抜き確認
R22196  ; ﾌﾗﾝｼﾞ穴検出下降停止遅延
R22208  ; ﾜｲﾊﾟｰ注油間欠吐出/待ち時間
R22209  ; ﾜｲﾊﾟｰ注油注油時間
R22234  ; ﾊﾞｯｸﾌﾞｰｽﾀ後退時間
R22353  ; ﾌﾗﾝｼﾞ穴検下降時間***A
R22354  ; 座屈検出監視時間
R22457  ; ﾊﾟｲﾌﾟ径ﾃﾞｰﾀ65A
R22458  ; ﾊﾟｲﾌﾟ径ﾃﾞｰﾀ80A
R22459  ; ﾊﾟｲﾌﾟ径ﾃﾞｰﾀ100A
R22472  ; 曲げＲ2.5D
R22473  ; 曲げＲ3.0D
R22474  ; 曲げＲ3.5D
R22475  ; 曲げＲ4.0D
R22476  ; 曲げＲ4.5D
R22477  ; 曲げＲ5.0D
R23561  ; BT2_CP2
R23562  ; BT2_CP3
R23563  ; BT2_CP4
R23564  ; BT2_CP5
R23565  ; BT2_CP6
R23566  ; BT2_CP7
R23567  ; BT2_CP8
R23568  ; BT2_CP9
R23569  ; BT2_CP10
R23571  ; BT3_CP2
R23572  ; BT3_CP3
R23573  ; BT3_CP4
R23574  ; BT3_CP5
R23575  ; BT3_CP6
R23576  ; BT3_CP7
R23577  ; BT3_CP8
R23578  ; BT3_CP9
R23579  ; BT3_CP10
R23581  ; BT4_CP2
R23582  ; BT4_CP3
R23583  ; BT4_CP4
R23584  ; BT4_CP5
R23585  ; BT4_CP6
R23586  ; BT4_CP7
R23587  ; BT4_CP8
R23588  ; BT4_CP9
R23589  ; BT4_CP10
R23590  ; BT5_CP1
R23591  ; BT5_CP2
R23592  ; BT5_CP3
R23593  ; BT5_CP4
R23594  ; BT5_CP5
R23595  ; BT5_CP6
R23596  ; BT5_CP7
R23597  ; BT5_CP8
R23598  ; BT5_CP9
R23599  ; BT5_CP10
R23600  ; BT6_CP1
R23601  ; BT6_CP2
R23602  ; BT6_CP3
R23603  ; BT6_CP4
R23604  ; BT6_CP5
R23605  ; BT6_CP6
R23606  ; BT6_CP7
R23607  ; BT6_CP8
R23608  ; BT6_CP9
R23609  ; BT6_CP10
R23610  ; BT7_CP1
R23611  ; BT7_CP2
R23612  ; BT7_CP3
R23613  ; BT7_CP4
R23614  ; BT7_CP5
R23615  ; BT7_CP6
R23616  ; BT7_CP7
R23617  ; BT7_CP8
R23618  ; BT7_CP9
R23619  ; BT7_CP10
R23620  ; BT8_CP1
R23621  ; BT8_CP2
R23622  ; BT8_CP3
R23623  ; BT8_CP4
R23624  ; BT8_CP5
R23625  ; BT8_CP6
R23626  ; BT8_CP7
R23627  ; BT8_CP8
R23628  ; BT8_CP9
R23629  ; BT8_CP10
R23661  ; BT2_BP2
R23662  ; BT2_BP3
R23663  ; BT2_BP4
R23664  ; BT2_BP5
R23665  ; BT2_BP6
R23666  ; BT2_BP7
R23667  ; BT2_BP8
R23668  ; BT2_BP9
R23669  ; BT2_BP10
R23671  ; BT3_BP2
R23672  ; BT3_BP3
R23673  ; BT3_BP4
R23674  ; BT3_BP5
R23675  ; BT3_BP6
R23676  ; BT3_BP7
R23677  ; BT3_BP8
R23678  ; BT3_BP9
R23679  ; BT3_BP10
R23681  ; BT4_BP2
R23682  ; BT4_BP3
R23683  ; BT4_BP4
R23684  ; BT4_BP5
R23685  ; BT4_BP6
R23686  ; BT4_BP7
R23687  ; BT4_BP8
R23688  ; BT4_BP9
R23689  ; BT4_BP10
R23690  ; BT5_BP1
R23691  ; BT5_BP2
R23692  ; BT5_BP3
R23693  ; BT5_BP4
R23694  ; BT5_BP5
R23695  ; BT5_BP6
R23696  ; BT5_BP7
R23697  ; BT5_BP8
R23698  ; BT5_BP9
R23699  ; BT5_BP10
R23700  ; BT6_BP1
R23701  ; BT6_BP2
R23702  ; BT6_BP3
R23703  ; BT6_BP4
R23704  ; BT6_BP5
R23705  ; BT6_BP6
R23706  ; BT6_BP7
R23707  ; BT6_BP8
R23708  ; BT6_BP9
R23709  ; BT6_BP10
R23710  ; BT7_BP1
R23711  ; BT7_BP2
R23712  ; BT7_BP3
R23713  ; BT7_BP4
R23714  ; BT7_BP5
R23715  ; BT7_BP6
R23716  ; BT7_BP7
R23717  ; BT7_BP8
R23718  ; BT7_BP9
R23719  ; BT7_BP10
R23720  ; BT8_BP1
R23721  ; BT8_BP2
R23722  ; BT8_BP3
R23723  ; BT8_BP4
R23724  ; BT8_BP5
R23725  ; BT8_BP6
R23726  ; BT8_BP7
R23727  ; BT8_BP8
R23728  ; BT8_BP9
R23729  ; BT8_BP10
R24050  ; 管番号_ＢＡ
R24091  ; 完了本数□□□本
R24100  ; 各種ﾃｰﾌﾞﾙNo.□□□
R24110  ; ﾌﾗﾝｼﾞ(ｸﾗﾝﾌﾟ側)_**k
R24114  ; ﾌﾗﾝｼﾞ(ﾁｬｯｸ側)_**k
R24350  ; Y軸曲げﾃﾞｰﾀ 1段
R24352  ; Y軸曲げﾃﾞｰﾀ 2段
R24354  ; Y軸曲げﾃﾞｰﾀ 3段
R24356  ; Y軸曲げﾃﾞｰﾀ 4段
R24358  ; Y軸曲げﾃﾞｰﾀ 5段
R24360  ; Y軸曲げﾃﾞｰﾀ 6段
R24362  ; Y軸曲げﾃﾞｰﾀ 7段
R24364  ; Y軸曲げﾃﾞｰﾀ 8段
R24366  ; Y軸曲げﾃﾞｰﾀ 9段
R24368  ; Y軸曲げﾃﾞｰﾀ 10段
R24370  ; Y軸曲げﾃﾞｰﾀ 11段
R24372  ; Y軸曲げﾃﾞｰﾀ 12段
R24374  ; Y軸曲げﾃﾞｰﾀ 13段
R24376  ; Y軸曲げﾃﾞｰﾀ 14段
R24378  ; Y軸曲げﾃﾞｰﾀ 15段
R24380  ; Y軸曲げﾃﾞｰﾀ 16段
R24382  ; Y軸曲げﾃﾞｰﾀ 17段
R24384  ; Y軸曲げﾃﾞｰﾀ 18段
R24386  ; Y軸曲げﾃﾞｰﾀ 19段
R24388  ; Y軸曲げﾃﾞｰﾀ 20段
R24390  ; Y軸曲げﾃﾞｰﾀ 21段
R24392  ; Y軸曲げﾃﾞｰﾀ 22段
R24394  ; Y軸曲げﾃﾞｰﾀ 23段
R24396  ; Y軸曲げﾃﾞｰﾀ 24段
R24398  ; Y軸曲げﾃﾞｰﾀ 25段
R24400  ; Y軸曲げﾃﾞｰﾀ 26段
R24402  ; Y軸曲げﾃﾞｰﾀ 27段
R24404  ; Y軸曲げﾃﾞｰﾀ 28段
R24406  ; Y軸曲げﾃﾞｰﾀ 29段
R24408  ; Y軸曲げﾃﾞｰﾀ 30段
R24420  ; B軸曲げﾃﾞｰﾀ 1段
R24422  ; B軸曲げﾃﾞｰﾀ 2段
R24424  ; B軸曲げﾃﾞｰﾀ 3段
R24426  ; B軸曲げﾃﾞｰﾀ 4段
R24428  ; B軸曲げﾃﾞｰﾀ 5段
R24430  ; B軸曲げﾃﾞｰﾀ 6段
R24432  ; B軸曲げﾃﾞｰﾀ 7段
R24434  ; B軸曲げﾃﾞｰﾀ 8段
R24436  ; B軸曲げﾃﾞｰﾀ 9段
R24438  ; B軸曲げﾃﾞｰﾀ10段
R24440  ; B軸曲げﾃﾞｰﾀ11段
R24442  ; B軸曲げﾃﾞｰﾀ12段
R24444  ; B軸曲げﾃﾞｰﾀ13段
R24446  ; B軸曲げﾃﾞｰﾀ14段
R24448  ; B軸曲げﾃﾞｰﾀ15段
R24450  ; B軸曲げﾃﾞｰﾀ16段
R24452  ; B軸曲げﾃﾞｰﾀ17段
R24454  ; B軸曲げﾃﾞｰﾀ18段
R24456  ; B軸曲げﾃﾞｰﾀ19段
R24458  ; B軸曲げﾃﾞｰﾀ20段
R24460  ; B軸曲げﾃﾞｰﾀ21段
R24462  ; B軸曲げﾃﾞｰﾀ22段
R24464  ; B軸曲げﾃﾞｰﾀ23段
R24466  ; B軸曲げﾃﾞｰﾀ24段
R24468  ; B軸曲げﾃﾞｰﾀ25段
R24470  ; B軸曲げﾃﾞｰﾀ26段
R24472  ; B軸曲げﾃﾞｰﾀ27段
R24474  ; B軸曲げﾃﾞｰﾀ28段
R24476  ; B軸曲げﾃﾞｰﾀ29段
R24478  ; B軸曲げﾃﾞｰﾀ30段
R24490  ; C軸曲げﾃﾞｰﾀ 1段
R24492  ; C軸曲げﾃﾞｰﾀ 2段
R24494  ; C軸曲げﾃﾞｰﾀ 3段
R24496  ; C軸曲げﾃﾞｰﾀ 4段
R24498  ; C軸曲げﾃﾞｰﾀ 5段
R24500  ; C軸曲げﾃﾞｰﾀ 6段
R24502  ; C軸曲げﾃﾞｰﾀ 7段
R24504  ; C軸曲げﾃﾞｰﾀ 8段
R24506  ; C軸曲げﾃﾞｰﾀ 9段
R24508  ; C軸曲げﾃﾞｰﾀ10段
R24510  ; C軸曲げﾃﾞｰﾀ11段
R24512  ; C軸曲げﾃﾞｰﾀ12段
R24514  ; C軸曲げﾃﾞｰﾀ13段
R24516  ; C軸曲げﾃﾞｰﾀ14段
R24518  ; C軸曲げﾃﾞｰﾀ15段
R24520  ; C軸曲げﾃﾞｰﾀ16段
R24522  ; C軸曲げﾃﾞｰﾀ17段
R24524  ; C軸曲げﾃﾞｰﾀ18段
R24526  ; C軸曲げﾃﾞｰﾀ19段
R24528  ; C軸曲げﾃﾞｰﾀ20段
R24530  ; C軸曲げﾃﾞｰﾀ21段
R24532  ; C軸曲げﾃﾞｰﾀ22段
R24534  ; C軸曲げﾃﾞｰﾀ23段
R24536  ; C軸曲げﾃﾞｰﾀ24段
R24538  ; C軸曲げﾃﾞｰﾀ25段
R24540  ; C軸曲げﾃﾞｰﾀ26段
R24542  ; C軸曲げﾃﾞｰﾀ27段
R24544  ; C軸曲げﾃﾞｰﾀ28段
R24546  ; C軸曲げﾃﾞｰﾀ29段
R24548  ; C軸曲げﾃﾞｰﾀ30段
R24665  ; Y軸ﾏｽﾀｰ曲げ 1段
R24667  ; Y軸ﾏｽﾀｰ曲げ 2段
R24669  ; Y軸ﾏｽﾀｰ曲げ 3段
R24671  ; Y軸ﾏｽﾀｰ曲げ 4段
R24673  ; Y軸ﾏｽﾀｰ曲げ 5段
R24675  ; Y軸ﾏｽﾀｰ曲げ 6段
R24677  ; Y軸ﾏｽﾀｰ曲げ 7段
R24679  ; Y軸ﾏｽﾀｰ曲げ 8段
R24681  ; Y軸ﾏｽﾀｰ曲げ 9段
R24683  ; Y軸ﾏｽﾀｰ曲げ10段
R24685  ; Y軸ﾏｽﾀｰ曲げ11段
R24687  ; Y軸ﾏｽﾀｰ曲げ12段
R24689  ; Y軸ﾏｽﾀｰ曲げ13段
R24691  ; Y軸ﾏｽﾀｰ曲げ14段
R24693  ; Y軸ﾏｽﾀｰ曲げ15段
R24695  ; Y軸ﾏｽﾀｰ曲げ16段
R24697  ; Y軸ﾏｽﾀｰ曲げ17段
R24699  ; Y軸ﾏｽﾀｰ曲げ18段
R24701  ; Y軸ﾏｽﾀｰ曲げ19段
R24703  ; Y軸ﾏｽﾀｰ曲げ20段
R24705  ; Y軸ﾏｽﾀｰ曲げ21段
R24707  ; Y軸ﾏｽﾀｰ曲げ22段
R24709  ; Y軸ﾏｽﾀｰ曲げ23段
R24711  ; Y軸ﾏｽﾀｰ曲げ24段
R24713  ; Y軸ﾏｽﾀｰ曲げ25段
R24715  ; Y軸ﾏｽﾀｰ曲げ26段
R24717  ; Y軸ﾏｽﾀｰ曲げ27段
R24719  ; Y軸ﾏｽﾀｰ曲げ28段
R24721  ; Y軸ﾏｽﾀｰ曲げ29段
R24723  ; Y軸ﾏｽﾀｰ曲げ30段
R24735  ; B軸ﾏｽﾀｰ曲げ 1段
R24737  ; B軸ﾏｽﾀｰ曲げ 2段
R24739  ; B軸ﾏｽﾀｰ曲げ 3段
R24741  ; B軸ﾏｽﾀｰ曲げ 4段
R24743  ; B軸ﾏｽﾀｰ曲げ 5段
R24745  ; B軸ﾏｽﾀｰ曲げ 6段
R24747  ; B軸ﾏｽﾀｰ曲げ 7段
R24749  ; B軸ﾏｽﾀｰ曲げ 8段
R24751  ; B軸ﾏｽﾀｰ曲げ 9段
R24753  ; B軸ﾏｽﾀｰ曲げ 10段
R24755  ; B軸ﾏｽﾀｰ曲げ 11段
R24757  ; B軸ﾏｽﾀｰ曲げ 12段
R24759  ; B軸ﾏｽﾀｰ曲げ 13段
R24761  ; B軸ﾏｽﾀｰ曲げ 14段
R24763  ; B軸ﾏｽﾀｰ曲げ 15段
R24765  ; B軸ﾏｽﾀｰ曲げ 16段
R24767  ; B軸ﾏｽﾀｰ曲げ 17段
R24769  ; B軸ﾏｽﾀｰ曲げ 18段
R24771  ; B軸ﾏｽﾀｰ曲げ 19段
R24773  ; B軸ﾏｽﾀｰ曲げ 20段
R24775  ; B軸ﾏｽﾀｰ曲げ 21段
R24777  ; B軸ﾏｽﾀｰ曲げ 22段
R24779  ; B軸ﾏｽﾀｰ曲げ 23段
R24781  ; B軸ﾏｽﾀｰ曲げ 24段
R24783  ; B軸ﾏｽﾀｰ曲げ 25段
R24785  ; B軸ﾏｽﾀｰ曲げ 26段
R24787  ; B軸ﾏｽﾀｰ曲げ 27段
R24789  ; B軸ﾏｽﾀｰ曲げ 28段
R24791  ; B軸ﾏｽﾀｰ曲げ 29段
R24793  ; B軸ﾏｽﾀｰ曲げ 30段
R24805  ; C軸ﾏｽﾀｰ曲げ 1段
R24807  ; C軸ﾏｽﾀｰ曲げ 2段
R24809  ; C軸ﾏｽﾀｰ曲げ 3段
R24811  ; C軸ﾏｽﾀｰ曲げ 4段
R24813  ; C軸ﾏｽﾀｰ曲げ 5段
R24815  ; C軸ﾏｽﾀｰ曲げ 6段
R24817  ; C軸ﾏｽﾀｰ曲げ 7段
R24819  ; C軸ﾏｽﾀｰ曲げ 8段
R24821  ; C軸ﾏｽﾀｰ曲げ 9段
R24823  ; C軸ﾏｽﾀｰ曲げ10段
R24825  ; C軸ﾏｽﾀｰ曲げ11段
R24827  ; C軸ﾏｽﾀｰ曲げ12段
R24829  ; C軸ﾏｽﾀｰ曲げ13段
R24831  ; C軸ﾏｽﾀｰ曲げ14段
R24833  ; C軸ﾏｽﾀｰ曲げ15段
R24835  ; C軸ﾏｽﾀｰ曲げ16段
R24837  ; C軸ﾏｽﾀｰ曲げ17段
R24839  ; C軸ﾏｽﾀｰ曲げ18段
R24841  ; C軸ﾏｽﾀｰ曲げ19段
R24843  ; C軸ﾏｽﾀｰ曲げ20段
R24845  ; C軸ﾏｽﾀｰ曲げ21段
R24847  ; C軸ﾏｽﾀｰ曲げ22段
R24849  ; C軸ﾏｽﾀｰ曲げ23段
R24851  ; C軸ﾏｽﾀｰ曲げ24段
R24853  ; C軸ﾏｽﾀｰ曲げ25段
R24855  ; C軸ﾏｽﾀｰ曲げ26段
R24857  ; C軸ﾏｽﾀｰ曲げ27段
R24859  ; C軸ﾏｽﾀｰ曲げ28段
R24861  ; C軸ﾏｽﾀｰ曲げ29段
R24863  ; C軸ﾏｽﾀｰ曲げ30段
ZR29000  ; 曲げﾜｰｸﾃﾞｰﾀ計算方法選択
ZR29001  ; ﾍﾟﾝﾀﾞﾝﾄ使用選択
ZR30050  ; 各種ﾃｰﾌﾞﾙNo.□□□
ZR30060  ; 始点金物_ＢＡ
ZR30061  ; 始点金物_ＤＣ
ZR30062  ; 始点金物_ＦＥ
ZR30063  ; 始点金物_ＨＧ
ZR30064  ; 終点金物_ＢＡ
ZR30065  ; 終点金物_ＤＣ
ZR30066  ; 終点金物_ＦＥ
ZR30067  ; 終点金物_ＨＧ
ZR30068  ; 始点金物出量_±□□.□mm
ZR30069  ; 終点金物出量_±□□.□mm
ZR30100  ; ﾊﾞｯｸﾌﾞｰｽﾀﾃｰﾌﾞﾙNo. 1段
ZR30101  ; ﾊﾞｯｸﾌﾞｰｽﾀﾃｰﾌﾞﾙNo. 2段
ZR30102  ; ﾊﾞｯｸﾌﾞｰｽﾀﾃｰﾌﾞﾙNo. 3段
ZR30103  ; ﾊﾞｯｸﾌﾞｰｽﾀﾃｰﾌﾞﾙNo. 4段
ZR30104  ; ﾊﾞｯｸﾌﾞｰｽﾀﾃｰﾌﾞﾙNo. 5段
ZR30105  ; ﾊﾞｯｸﾌﾞｰｽﾀﾃｰﾌﾞﾙNo. 6段
ZR30106  ; ﾊﾞｯｸﾌﾞｰｽﾀﾃｰﾌﾞﾙNo. 7段
ZR30107  ; ﾊﾞｯｸﾌﾞｰｽﾀﾃｰﾌﾞﾙNo. 8段
ZR30108  ; ﾊﾞｯｸﾌﾞｰｽﾀﾃｰﾌﾞﾙNo. 9段
ZR30109  ; ﾊﾞｯｸﾌﾞｰｽﾀﾃｰﾌﾞﾙNo. 10段
ZR30110  ; ﾊﾞｯｸﾌﾞｰｽﾀﾃｰﾌﾞﾙNo. 11段
ZR30111  ; ﾊﾞｯｸﾌﾞｰｽﾀﾃｰﾌﾞﾙNo. 12段
ZR30112  ; ﾊﾞｯｸﾌﾞｰｽﾀﾃｰﾌﾞﾙNo. 13段
ZR30113  ; ﾊﾞｯｸﾌﾞｰｽﾀﾃｰﾌﾞﾙNo. 14段
ZR30114  ; ﾊﾞｯｸﾌﾞｰｽﾀﾃｰﾌﾞﾙNo. 15段
ZR30115  ; ﾊﾞｯｸﾌﾞｰｽﾀﾃｰﾌﾞﾙNo. 16段
ZR30116  ; ﾊﾞｯｸﾌﾞｰｽﾀﾃｰﾌﾞﾙNo. 17段
ZR30117  ; ﾊﾞｯｸﾌﾞｰｽﾀﾃｰﾌﾞﾙNo. 18段
ZR30118  ; ﾊﾞｯｸﾌﾞｰｽﾀﾃｰﾌﾞﾙNo. 19段
ZR30119  ; ﾊﾞｯｸﾌﾞｰｽﾀﾃｰﾌﾞﾙNo. 20段
ZR30120  ; ﾊﾞｯｸﾌﾞｰｽﾀﾃｰﾌﾞﾙNo. 21段
ZR30121  ; ﾊﾞｯｸﾌﾞｰｽﾀﾃｰﾌﾞﾙNo. 22段
ZR30122  ; ﾊﾞｯｸﾌﾞｰｽﾀﾃｰﾌﾞﾙNo. 23段
ZR30123  ; ﾊﾞｯｸﾌﾞｰｽﾀﾃｰﾌﾞﾙNo. 24段
ZR30124  ; ﾊﾞｯｸﾌﾞｰｽﾀﾃｰﾌﾞﾙNo. 25段
ZR30125  ; ﾊﾞｯｸﾌﾞｰｽﾀﾃｰﾌﾞﾙNo. 26段
ZR30126  ; ﾊﾞｯｸﾌﾞｰｽﾀﾃｰﾌﾞﾙNo. 27段
ZR30127  ; ﾊﾞｯｸﾌﾞｰｽﾀﾃｰﾌﾞﾙNo. 28段
ZR30128  ; ﾊﾞｯｸﾌﾞｰｽﾀﾃｰﾌﾞﾙNo. 29段
ZR30129  ; ﾊﾞｯｸﾌﾞｰｽﾀﾃｰﾌﾞﾙNo. 30段
ZR30300  ; Y軸ﾏｽﾀﾃﾞｰﾀ 1段
ZR30302  ; Y軸ﾏｽﾀﾃﾞｰﾀ 2段
ZR30304  ; Y軸ﾏｽﾀﾃﾞｰﾀ 3段
ZR30306  ; Y軸ﾏｽﾀﾃﾞｰﾀ 4段
ZR30308  ; Y軸ﾏｽﾀﾃﾞｰﾀ 5段
ZR30310  ; Y軸ﾏｽﾀﾃﾞｰﾀ 6段
ZR30312  ; Y軸ﾏｽﾀﾃﾞｰﾀ 7段
ZR30314  ; Y軸ﾏｽﾀﾃﾞｰﾀ 8段
ZR30316  ; Y軸ﾏｽﾀﾃﾞｰﾀ 9段
ZR30318  ; Y軸ﾏｽﾀﾃﾞｰﾀ 10段
ZR30320  ; Y軸ﾏｽﾀﾃﾞｰﾀ 11段
ZR30322  ; Y軸ﾏｽﾀﾃﾞｰﾀ 12段
ZR30324  ; Y軸ﾏｽﾀﾃﾞｰﾀ 13段
ZR30326  ; Y軸ﾏｽﾀﾃﾞｰﾀ 14段
ZR30328  ; Y軸ﾏｽﾀﾃﾞｰﾀ 15段
ZR30330  ; Y軸ﾏｽﾀﾃﾞｰﾀ 16段
ZR30332  ; Y軸ﾏｽﾀﾃﾞｰﾀ 17段
ZR30334  ; Y軸ﾏｽﾀﾃﾞｰﾀ 18段
ZR30336  ; Y軸ﾏｽﾀﾃﾞｰﾀ 19段
ZR30338  ; Y軸ﾏｽﾀﾃﾞｰﾀ 20段
ZR30340  ; Y軸ﾏｽﾀﾃﾞｰﾀ 21段
ZR30342  ; Y軸ﾏｽﾀﾃﾞｰﾀ 22段
ZR30344  ; Y軸ﾏｽﾀﾃﾞｰﾀ 23段
ZR30346  ; Y軸ﾏｽﾀﾃﾞｰﾀ 24段
ZR30348  ; Y軸ﾏｽﾀﾃﾞｰﾀ 25段
ZR30350  ; Y軸ﾏｽﾀﾃﾞｰﾀ 26段
ZR30352  ; Y軸ﾏｽﾀﾃﾞｰﾀ 27段
ZR30354  ; Y軸ﾏｽﾀﾃﾞｰﾀ 28段
ZR30356  ; Y軸ﾏｽﾀﾃﾞｰﾀ 29段
ZR30358  ; Y軸ﾏｽﾀﾃﾞｰﾀ 30段
ZR30370  ; B軸ﾏｽﾀﾃﾞｰﾀ 1段
ZR30372  ; B軸ﾏｽﾀﾃﾞｰﾀ 2段
ZR30374  ; B軸ﾏｽﾀﾃﾞｰﾀ 3段
ZR30376  ; B軸ﾏｽﾀﾃﾞｰﾀ 4段
ZR30378  ; B軸ﾏｽﾀﾃﾞｰﾀ 5段
ZR30380  ; B軸ﾏｽﾀﾃﾞｰﾀ 6段
ZR30382  ; B軸ﾏｽﾀﾃﾞｰﾀ 7段
ZR30384  ; B軸ﾏｽﾀﾃﾞｰﾀ 8段
ZR30386  ; B軸ﾏｽﾀﾃﾞｰﾀ 9段
ZR30388  ; B軸ﾏｽﾀﾃﾞｰﾀ10段
ZR30390  ; B軸ﾏｽﾀﾃﾞｰﾀ11段
ZR30392  ; B軸ﾏｽﾀﾃﾞｰﾀ12段
ZR30394  ; B軸ﾏｽﾀﾃﾞｰﾀ13段
ZR30396  ; B軸ﾏｽﾀﾃﾞｰﾀ14段
ZR30398  ; B軸ﾏｽﾀﾃﾞｰﾀ15段
ZR30400  ; B軸ﾏｽﾀﾃﾞｰﾀ16段
ZR30402  ; B軸ﾏｽﾀﾃﾞｰﾀ17段
ZR30404  ; B軸ﾏｽﾀﾃﾞｰﾀ18段
ZR30406  ; B軸ﾏｽﾀﾃﾞｰﾀ19段
ZR30408  ; B軸ﾏｽﾀﾃﾞｰﾀ20段
ZR30410  ; B軸ﾏｽﾀﾃﾞｰﾀ21段
ZR30412  ; B軸ﾏｽﾀﾃﾞｰﾀ22段
ZR30414  ; B軸ﾏｽﾀﾃﾞｰﾀ23段
ZR30416  ; B軸ﾏｽﾀﾃﾞｰﾀ24段
ZR30418  ; B軸ﾏｽﾀﾃﾞｰﾀ25段
ZR30420  ; B軸ﾏｽﾀﾃﾞｰﾀ26段
ZR30422  ; B軸ﾏｽﾀﾃﾞｰﾀ27段
ZR30424  ; B軸ﾏｽﾀﾃﾞｰﾀ28段
ZR30426  ; B軸ﾏｽﾀﾃﾞｰﾀ29段
ZR30428  ; B軸ﾏｽﾀﾃﾞｰﾀ30段
ZR30440  ; C軸ﾏｽﾀﾃﾞｰﾀ 1段
ZR30442  ; C軸ﾏｽﾀﾃﾞｰﾀ 2段
ZR30444  ; C軸ﾏｽﾀﾃﾞｰﾀ 3段
ZR30446  ; C軸ﾏｽﾀﾃﾞｰﾀ 4段
ZR30448  ; C軸ﾏｽﾀﾃﾞｰﾀ 5段
ZR30450  ; C軸ﾏｽﾀﾃﾞｰﾀ 6段
ZR30452  ; C軸ﾏｽﾀﾃﾞｰﾀ 7段
ZR30454  ; C軸ﾏｽﾀﾃﾞｰﾀ 8段
ZR30456  ; C軸ﾏｽﾀﾃﾞｰﾀ 9段
ZR30458  ; C軸ﾏｽﾀﾃﾞｰﾀ10段
ZR30460  ; C軸ﾏｽﾀﾃﾞｰﾀ11段
ZR30462  ; C軸ﾏｽﾀﾃﾞｰﾀ12段
ZR30464  ; C軸ﾏｽﾀﾃﾞｰﾀ13段
ZR30466  ; C軸ﾏｽﾀﾃﾞｰﾀ14段
ZR30468  ; C軸ﾏｽﾀﾃﾞｰﾀ15段
ZR30470  ; C軸ﾏｽﾀﾃﾞｰﾀ16段
ZR30472  ; C軸ﾏｽﾀﾃﾞｰﾀ17段
ZR30474  ; C軸ﾏｽﾀﾃﾞｰﾀ18段
ZR30476  ; C軸ﾏｽﾀﾃﾞｰﾀ19段
ZR30478  ; C軸ﾏｽﾀﾃﾞｰﾀ20段
ZR30480  ; C軸ﾏｽﾀﾃﾞｰﾀ21段
ZR30482  ; C軸ﾏｽﾀﾃﾞｰﾀ22段
ZR30484  ; C軸ﾏｽﾀﾃﾞｰﾀ23段
ZR30486  ; C軸ﾏｽﾀﾃﾞｰﾀ24段
ZR30488  ; C軸ﾏｽﾀﾃﾞｰﾀ25段
ZR30490  ; C軸ﾏｽﾀﾃﾞｰﾀ26段
ZR30492  ; C軸ﾏｽﾀﾃﾞｰﾀ27段
ZR30494  ; C軸ﾏｽﾀﾃﾞｰﾀ28段
ZR30496  ; C軸ﾏｽﾀﾃﾞｰﾀ29段
ZR30498  ; C軸ﾏｽﾀﾃﾞｰﾀ30段
ZR30615  ; Y軸ﾜｰｸ曲げﾃﾞｰﾀ 1段
ZR30617  ; Y軸ﾜｰｸ曲げﾃﾞｰﾀ 2段
ZR30619  ; Y軸ﾜｰｸ曲げﾃﾞｰﾀ 3段
ZR30621  ; Y軸ﾜｰｸ曲げﾃﾞｰﾀ 4段
ZR30623  ; Y軸ﾜｰｸ曲げﾃﾞｰﾀ 5段
ZR30625  ; Y軸ﾜｰｸ曲げﾃﾞｰﾀ 6段
ZR30627  ; Y軸ﾜｰｸ曲げﾃﾞｰﾀ 7段
ZR30629  ; Y軸ﾜｰｸ曲げﾃﾞｰﾀ 8段
ZR30631  ; Y軸ﾜｰｸ曲げﾃﾞｰﾀ 9段
ZR30633  ; Y軸ﾜｰｸ曲げﾃﾞｰﾀ10段
ZR30635  ; Y軸ﾜｰｸ曲げﾃﾞｰﾀ11段
ZR30637  ; Y軸ﾜｰｸ曲げﾃﾞｰﾀ12段
ZR30639  ; Y軸ﾜｰｸ曲げﾃﾞｰﾀ13段
ZR30641  ; Y軸ﾜｰｸ曲げﾃﾞｰﾀ14段
ZR30643  ; Y軸ﾜｰｸ曲げﾃﾞｰﾀ15段
ZR30645  ; Y軸ﾜｰｸ曲げﾃﾞｰﾀ16段
ZR30647  ; Y軸ﾜｰｸ曲げﾃﾞｰﾀ17段
ZR30649  ; Y軸ﾜｰｸ曲げﾃﾞｰﾀ18段
ZR30651  ; Y軸ﾜｰｸ曲げﾃﾞｰﾀ19段
ZR30653  ; Y軸ﾜｰｸ曲げﾃﾞｰﾀ20段
ZR30655  ; Y軸ﾜｰｸ曲げﾃﾞｰﾀ21段
ZR30657  ; Y軸ﾜｰｸ曲げﾃﾞｰﾀ22段
ZR30659  ; Y軸ﾜｰｸ曲げﾃﾞｰﾀ23段
ZR30661  ; Y軸ﾜｰｸ曲げﾃﾞｰﾀ24段
ZR30663  ; Y軸ﾜｰｸ曲げﾃﾞｰﾀ25段
ZR30665  ; Y軸ﾜｰｸ曲げﾃﾞｰﾀ26段
ZR30667  ; Y軸ﾜｰｸ曲げﾃﾞｰﾀ27段
ZR30669  ; Y軸ﾜｰｸ曲げﾃﾞｰﾀ28段
ZR30671  ; Y軸ﾜｰｸ曲げﾃﾞｰﾀ29段
ZR30673  ; Y軸ﾜｰｸ曲げﾃﾞｰﾀ30段
ZR30685  ; B軸ﾜｰｸ曲げﾃﾞｰﾀ 1段
ZR30687  ; B軸ﾜｰｸ曲げﾃﾞｰﾀ 2段
ZR30689  ; B軸ﾜｰｸ曲げﾃﾞｰﾀ 3段
ZR30691  ; B軸ﾜｰｸ曲げﾃﾞｰﾀ 4段
ZR30693  ; B軸ﾜｰｸ曲げﾃﾞｰﾀ 5段
ZR30695  ; B軸ﾜｰｸ曲げﾃﾞｰﾀ 6段
ZR30697  ; B軸ﾜｰｸ曲げﾃﾞｰﾀ 7段
ZR30699  ; B軸ﾜｰｸ曲げﾃﾞｰﾀ 8段
ZR30701  ; B軸ﾜｰｸ曲げﾃﾞｰﾀ 9段
ZR30703  ; B軸ﾜｰｸ曲げﾃﾞｰﾀ 10段
ZR30705  ; B軸ﾜｰｸ曲げﾃﾞｰﾀ 11段
ZR30707  ; B軸ﾜｰｸ曲げﾃﾞｰﾀ 12段
ZR30709  ; B軸ﾜｰｸ曲げﾃﾞｰﾀ 13段
ZR30711  ; B軸ﾜｰｸ曲げﾃﾞｰﾀ 14段
ZR30713  ; B軸ﾜｰｸ曲げﾃﾞｰﾀ 15段
ZR30715  ; B軸ﾜｰｸ曲げﾃﾞｰﾀ 16段
ZR30717  ; B軸ﾜｰｸ曲げﾃﾞｰﾀ 17段
ZR30719  ; B軸ﾜｰｸ曲げﾃﾞｰﾀ 18段
ZR30721  ; B軸ﾜｰｸ曲げﾃﾞｰﾀ 19段
ZR30723  ; B軸ﾜｰｸ曲げﾃﾞｰﾀ 20段
ZR30725  ; B軸ﾜｰｸ曲げﾃﾞｰﾀ 21段
ZR30727  ; B軸ﾜｰｸ曲げﾃﾞｰﾀ 22段
ZR30729  ; B軸ﾜｰｸ曲げﾃﾞｰﾀ 23段
ZR30731  ; B軸ﾜｰｸ曲げﾃﾞｰﾀ 24段
ZR30733  ; B軸ﾜｰｸ曲げﾃﾞｰﾀ 25段
ZR30735  ; B軸ﾜｰｸ曲げﾃﾞｰﾀ 26段
ZR30737  ; B軸ﾜｰｸ曲げﾃﾞｰﾀ 27段
ZR30739  ; B軸ﾜｰｸ曲げﾃﾞｰﾀ 28段
ZR30741  ; B軸ﾜｰｸ曲げﾃﾞｰﾀ 29段
ZR30743  ; B軸ﾜｰｸ曲げﾃﾞｰﾀ 30段
ZR30755  ; C軸ﾜｰｸ曲げﾃﾞｰﾀ 1段
ZR30757  ; C軸ﾜｰｸ曲げﾃﾞｰﾀ 2段
ZR30759  ; C軸ﾜｰｸ曲げﾃﾞｰﾀ 3段
ZR30761  ; C軸ﾜｰｸ曲げﾃﾞｰﾀ 4段
ZR30763  ; C軸ﾜｰｸ曲げﾃﾞｰﾀ 5段
ZR30765  ; C軸ﾜｰｸ曲げﾃﾞｰﾀ 6段
ZR30767  ; C軸ﾜｰｸ曲げﾃﾞｰﾀ 7段
ZR30769  ; C軸ﾜｰｸ曲げﾃﾞｰﾀ 8段
ZR30771  ; C軸ﾜｰｸ曲げﾃﾞｰﾀ 9段
ZR30773  ; C軸ﾜｰｸ曲げﾃﾞｰﾀ10段
ZR30775  ; C軸ﾜｰｸ曲げﾃﾞｰﾀ11段
ZR30777  ; C軸ﾜｰｸ曲げﾃﾞｰﾀ12段
ZR30779  ; C軸ﾜｰｸ曲げﾃﾞｰﾀ13段
ZR30781  ; C軸ﾜｰｸ曲げﾃﾞｰﾀ14段
ZR30783  ; C軸ﾜｰｸ曲げﾃﾞｰﾀ15段
ZR30785  ; C軸ﾜｰｸ曲げﾃﾞｰﾀ16段
ZR30787  ; C軸ﾜｰｸ曲げﾃﾞｰﾀ17段
ZR30789  ; C軸ﾜｰｸ曲げﾃﾞｰﾀ18段
ZR30791  ; C軸ﾜｰｸ曲げﾃﾞｰﾀ19段
ZR30793  ; C軸ﾜｰｸ曲げﾃﾞｰﾀ20段
ZR30795  ; C軸ﾜｰｸ曲げﾃﾞｰﾀ21段
ZR30797  ; C軸ﾜｰｸ曲げﾃﾞｰﾀ22段
ZR30799  ; C軸ﾜｰｸ曲げﾃﾞｰﾀ23段
ZR30801  ; C軸ﾜｰｸ曲げﾃﾞｰﾀ24段
ZR30803  ; C軸ﾜｰｸ曲げﾃﾞｰﾀ25段
ZR30805  ; C軸ﾜｰｸ曲げﾃﾞｰﾀ26段
ZR30807  ; C軸ﾜｰｸ曲げﾃﾞｰﾀ27段
ZR30809  ; C軸ﾜｰｸ曲げﾃﾞｰﾀ28段
ZR30811  ; C軸ﾜｰｸ曲げﾃﾞｰﾀ29段
ZR30813  ; C軸ﾜｰｸ曲げﾃﾞｰﾀ30段
ZR60041  ; 完了本数□□□本
ZR60300  ; Y軸ﾏｽﾀﾃﾞｰﾀ 1段
ZR60302  ; Y軸ﾏｽﾀﾃﾞｰﾀ 2段
ZR60304  ; Y軸ﾏｽﾀﾃﾞｰﾀ 3段
ZR60306  ; Y軸ﾏｽﾀﾃﾞｰﾀ 4段
ZR60308  ; Y軸ﾏｽﾀﾃﾞｰﾀ 5段
ZR60310  ; Y軸ﾏｽﾀﾃﾞｰﾀ 6段
ZR60312  ; Y軸ﾏｽﾀﾃﾞｰﾀ 7段
ZR60314  ; Y軸ﾏｽﾀﾃﾞｰﾀ 8段
ZR60316  ; Y軸ﾏｽﾀﾃﾞｰﾀ 9段
ZR60318  ; Y軸ﾏｽﾀﾃﾞｰﾀ 10段
ZR60320  ; Y軸ﾏｽﾀﾃﾞｰﾀ 11段
ZR60322  ; Y軸ﾏｽﾀﾃﾞｰﾀ 12段
ZR60324  ; Y軸ﾏｽﾀﾃﾞｰﾀ 13段
ZR60326  ; Y軸ﾏｽﾀﾃﾞｰﾀ 14段
ZR60328  ; Y軸ﾏｽﾀﾃﾞｰﾀ 15段
ZR60330  ; Y軸ﾏｽﾀﾃﾞｰﾀ 16段
ZR60332  ; Y軸ﾏｽﾀﾃﾞｰﾀ 17段
ZR60334  ; Y軸ﾏｽﾀﾃﾞｰﾀ 18段
ZR60336  ; Y軸ﾏｽﾀﾃﾞｰﾀ 19段
ZR60338  ; Y軸ﾏｽﾀﾃﾞｰﾀ 20段
ZR60340  ; Y軸ﾏｽﾀﾃﾞｰﾀ 21段
ZR60342  ; Y軸ﾏｽﾀﾃﾞｰﾀ 22段
ZR60344  ; Y軸ﾏｽﾀﾃﾞｰﾀ 23段
ZR60346  ; Y軸ﾏｽﾀﾃﾞｰﾀ 24段
ZR60348  ; Y軸ﾏｽﾀﾃﾞｰﾀ 25段
ZR60350  ; Y軸ﾏｽﾀﾃﾞｰﾀ 26段
ZR60352  ; Y軸ﾏｽﾀﾃﾞｰﾀ 27段
ZR60354  ; Y軸ﾏｽﾀﾃﾞｰﾀ 28段
ZR60356  ; Y軸ﾏｽﾀﾃﾞｰﾀ 29段
ZR60358  ; Y軸ﾏｽﾀﾃﾞｰﾀ 30段
ZR60370  ; B軸ﾏｽﾀﾃﾞｰﾀ 1段
ZR60372  ; B軸ﾏｽﾀﾃﾞｰﾀ 2段
ZR60374  ; B軸ﾏｽﾀﾃﾞｰﾀ 3段
ZR60376  ; B軸ﾏｽﾀﾃﾞｰﾀ 4段
ZR60378  ; B軸ﾏｽﾀﾃﾞｰﾀ 5段
ZR60380  ; B軸ﾏｽﾀﾃﾞｰﾀ 6段
ZR60382  ; B軸ﾏｽﾀﾃﾞｰﾀ 7段
ZR60384  ; B軸ﾏｽﾀﾃﾞｰﾀ 8段
ZR60386  ; B軸ﾏｽﾀﾃﾞｰﾀ 9段
ZR60388  ; B軸ﾏｽﾀﾃﾞｰﾀ10段
ZR60390  ; B軸ﾏｽﾀﾃﾞｰﾀ11段
ZR60392  ; B軸ﾏｽﾀﾃﾞｰﾀ12段
ZR60394  ; B軸ﾏｽﾀﾃﾞｰﾀ13段
ZR60396  ; B軸ﾏｽﾀﾃﾞｰﾀ14段
ZR60398  ; B軸ﾏｽﾀﾃﾞｰﾀ15段
ZR60400  ; B軸ﾏｽﾀﾃﾞｰﾀ16段
ZR60402  ; B軸ﾏｽﾀﾃﾞｰﾀ17段
ZR60404  ; B軸ﾏｽﾀﾃﾞｰﾀ18段
ZR60406  ; B軸ﾏｽﾀﾃﾞｰﾀ19段
ZR60408  ; B軸ﾏｽﾀﾃﾞｰﾀ20段
ZR60410  ; B軸ﾏｽﾀﾃﾞｰﾀ21段
ZR60412  ; B軸ﾏｽﾀﾃﾞｰﾀ22段
ZR60414  ; B軸ﾏｽﾀﾃﾞｰﾀ23段
ZR60416  ; B軸ﾏｽﾀﾃﾞｰﾀ24段
ZR60418  ; B軸ﾏｽﾀﾃﾞｰﾀ25段
ZR60420  ; B軸ﾏｽﾀﾃﾞｰﾀ26段
ZR60422  ; B軸ﾏｽﾀﾃﾞｰﾀ27段
ZR60424  ; B軸ﾏｽﾀﾃﾞｰﾀ28段
ZR60426  ; B軸ﾏｽﾀﾃﾞｰﾀ29段
ZR60428  ; B軸ﾏｽﾀﾃﾞｰﾀ30段
ZR60440  ; C軸ﾏｽﾀﾃﾞｰﾀ 1段
ZR60442  ; C軸ﾏｽﾀﾃﾞｰﾀ 2段
ZR60444  ; C軸ﾏｽﾀﾃﾞｰﾀ 3段
ZR60446  ; C軸ﾏｽﾀﾃﾞｰﾀ 4段
ZR60448  ; C軸ﾏｽﾀﾃﾞｰﾀ 5段
ZR60450  ; C軸ﾏｽﾀﾃﾞｰﾀ 6段
ZR60452  ; C軸ﾏｽﾀﾃﾞｰﾀ 7段
ZR60454  ; C軸ﾏｽﾀﾃﾞｰﾀ 8段
ZR60456  ; C軸ﾏｽﾀﾃﾞｰﾀ 9段
ZR60458  ; C軸ﾏｽﾀﾃﾞｰﾀ10段
ZR60460  ; C軸ﾏｽﾀﾃﾞｰﾀ11段
ZR60462  ; C軸ﾏｽﾀﾃﾞｰﾀ12段
ZR60464  ; C軸ﾏｽﾀﾃﾞｰﾀ13段
ZR60466  ; C軸ﾏｽﾀﾃﾞｰﾀ14段
ZR60468  ; C軸ﾏｽﾀﾃﾞｰﾀ15段
ZR60470  ; C軸ﾏｽﾀﾃﾞｰﾀ16段
ZR60472  ; C軸ﾏｽﾀﾃﾞｰﾀ17段
ZR60474  ; C軸ﾏｽﾀﾃﾞｰﾀ18段
ZR60476  ; C軸ﾏｽﾀﾃﾞｰﾀ19段
ZR60478  ; C軸ﾏｽﾀﾃﾞｰﾀ20段
ZR60480  ; C軸ﾏｽﾀﾃﾞｰﾀ21段
ZR60482  ; C軸ﾏｽﾀﾃﾞｰﾀ22段
ZR60484  ; C軸ﾏｽﾀﾃﾞｰﾀ23段
ZR60486  ; C軸ﾏｽﾀﾃﾞｰﾀ24段
ZR60488  ; C軸ﾏｽﾀﾃﾞｰﾀ25段
ZR60490  ; C軸ﾏｽﾀﾃﾞｰﾀ26段
ZR60492  ; C軸ﾏｽﾀﾃﾞｰﾀ27段
ZR60494  ; C軸ﾏｽﾀﾃﾞｰﾀ28段
ZR60496  ; C軸ﾏｽﾀﾃﾞｰﾀ29段
ZR60498  ; C軸ﾏｽﾀﾃﾞｰﾀ30段
ZR60615  ; Y軸ﾜｰｸ曲げﾃﾞｰﾀ 1段
ZR60617  ; Y軸ﾜｰｸ曲げﾃﾞｰﾀ 2段
ZR60619  ; Y軸ﾜｰｸ曲げﾃﾞｰﾀ 3段
ZR60621  ; Y軸ﾜｰｸ曲げﾃﾞｰﾀ 4段
ZR60623  ; Y軸ﾜｰｸ曲げﾃﾞｰﾀ 5段
ZR60625  ; Y軸ﾜｰｸ曲げﾃﾞｰﾀ 6段
ZR60627  ; Y軸ﾜｰｸ曲げﾃﾞｰﾀ 7段
ZR60629  ; Y軸ﾜｰｸ曲げﾃﾞｰﾀ 8段
ZR60631  ; Y軸ﾜｰｸ曲げﾃﾞｰﾀ 9段
ZR60633  ; Y軸ﾜｰｸ曲げﾃﾞｰﾀ10段
ZR60635  ; Y軸ﾜｰｸ曲げﾃﾞｰﾀ11段
ZR60637  ; Y軸ﾜｰｸ曲げﾃﾞｰﾀ12段
ZR60639  ; Y軸ﾜｰｸ曲げﾃﾞｰﾀ13段
ZR60641  ; Y軸ﾜｰｸ曲げﾃﾞｰﾀ14段
ZR60643  ; Y軸ﾜｰｸ曲げﾃﾞｰﾀ15段
ZR60645  ; Y軸ﾜｰｸ曲げﾃﾞｰﾀ16段
ZR60647  ; Y軸ﾜｰｸ曲げﾃﾞｰﾀ17段
ZR60649  ; Y軸ﾜｰｸ曲げﾃﾞｰﾀ18段
ZR60651  ; Y軸ﾜｰｸ曲げﾃﾞｰﾀ19段
ZR60653  ; Y軸ﾜｰｸ曲げﾃﾞｰﾀ20段
ZR60655  ; Y軸ﾜｰｸ曲げﾃﾞｰﾀ21段
ZR60657  ; Y軸ﾜｰｸ曲げﾃﾞｰﾀ22段
ZR60659  ; Y軸ﾜｰｸ曲げﾃﾞｰﾀ23段
ZR60661  ; Y軸ﾜｰｸ曲げﾃﾞｰﾀ24段
ZR60663  ; Y軸ﾜｰｸ曲げﾃﾞｰﾀ25段
ZR60665  ; Y軸ﾜｰｸ曲げﾃﾞｰﾀ26段
ZR60667  ; Y軸ﾜｰｸ曲げﾃﾞｰﾀ27段
ZR60669  ; Y軸ﾜｰｸ曲げﾃﾞｰﾀ28段
ZR60671  ; Y軸ﾜｰｸ曲げﾃﾞｰﾀ29段
ZR60673  ; Y軸ﾜｰｸ曲げﾃﾞｰﾀ30段
ZR60685  ; B軸ﾜｰｸ曲げﾃﾞｰﾀ 1段
ZR60687  ; B軸ﾜｰｸ曲げﾃﾞｰﾀ 2段
ZR60689  ; B軸ﾜｰｸ曲げﾃﾞｰﾀ 3段
ZR60691  ; B軸ﾜｰｸ曲げﾃﾞｰﾀ 4段
ZR60693  ; B軸ﾜｰｸ曲げﾃﾞｰﾀ 5段
ZR60695  ; B軸ﾜｰｸ曲げﾃﾞｰﾀ 6段
ZR60697  ; B軸ﾜｰｸ曲げﾃﾞｰﾀ 7段
ZR60699  ; B軸ﾜｰｸ曲げﾃﾞｰﾀ 8段
ZR60701  ; B軸ﾜｰｸ曲げﾃﾞｰﾀ 9段
ZR60703  ; B軸ﾜｰｸ曲げﾃﾞｰﾀ 10段
ZR60705  ; B軸ﾜｰｸ曲げﾃﾞｰﾀ 11段
ZR60707  ; B軸ﾜｰｸ曲げﾃﾞｰﾀ 12段
ZR60709  ; B軸ﾜｰｸ曲げﾃﾞｰﾀ 13段
ZR60711  ; B軸ﾜｰｸ曲げﾃﾞｰﾀ 14段
ZR60713  ; B軸ﾜｰｸ曲げﾃﾞｰﾀ 15段
ZR60715  ; B軸ﾜｰｸ曲げﾃﾞｰﾀ 16段
ZR60717  ; B軸ﾜｰｸ曲げﾃﾞｰﾀ 17段
ZR60719  ; B軸ﾜｰｸ曲げﾃﾞｰﾀ 18段
ZR60721  ; B軸ﾜｰｸ曲げﾃﾞｰﾀ 19段
ZR60723  ; B軸ﾜｰｸ曲げﾃﾞｰﾀ 20段
ZR60725  ; B軸ﾜｰｸ曲げﾃﾞｰﾀ 21段
ZR60727  ; B軸ﾜｰｸ曲げﾃﾞｰﾀ 22段
ZR60729  ; B軸ﾜｰｸ曲げﾃﾞｰﾀ 23段
ZR60731  ; B軸ﾜｰｸ曲げﾃﾞｰﾀ 24段
ZR60733  ; B軸ﾜｰｸ曲げﾃﾞｰﾀ 25段
ZR60735  ; B軸ﾜｰｸ曲げﾃﾞｰﾀ 26段
ZR60737  ; B軸ﾜｰｸ曲げﾃﾞｰﾀ 27段
ZR60739  ; B軸ﾜｰｸ曲げﾃﾞｰﾀ 28段
ZR60741  ; B軸ﾜｰｸ曲げﾃﾞｰﾀ 29段
ZR60743  ; B軸ﾜｰｸ曲げﾃﾞｰﾀ 30段
ZR60755  ; C軸ﾜｰｸ曲げﾃﾞｰﾀ 1段
ZR60757  ; C軸ﾜｰｸ曲げﾃﾞｰﾀ 2段
ZR60759  ; C軸ﾜｰｸ曲げﾃﾞｰﾀ 3段
ZR60761  ; C軸ﾜｰｸ曲げﾃﾞｰﾀ 4段
ZR60763  ; C軸ﾜｰｸ曲げﾃﾞｰﾀ 5段
ZR60765  ; C軸ﾜｰｸ曲げﾃﾞｰﾀ 6段
ZR60767  ; C軸ﾜｰｸ曲げﾃﾞｰﾀ 7段
ZR60769  ; C軸ﾜｰｸ曲げﾃﾞｰﾀ 8段
ZR60771  ; C軸ﾜｰｸ曲げﾃﾞｰﾀ 9段
ZR60773  ; C軸ﾜｰｸ曲げﾃﾞｰﾀ10段
ZR60775  ; C軸ﾜｰｸ曲げﾃﾞｰﾀ11段
ZR60777  ; C軸ﾜｰｸ曲げﾃﾞｰﾀ12段
ZR60779  ; C軸ﾜｰｸ曲げﾃﾞｰﾀ13段
ZR60781  ; C軸ﾜｰｸ曲げﾃﾞｰﾀ14段
ZR60783  ; C軸ﾜｰｸ曲げﾃﾞｰﾀ15段
ZR60785  ; C軸ﾜｰｸ曲げﾃﾞｰﾀ16段
ZR60787  ; C軸ﾜｰｸ曲げﾃﾞｰﾀ17段
ZR60789  ; C軸ﾜｰｸ曲げﾃﾞｰﾀ18段
ZR60791  ; C軸ﾜｰｸ曲げﾃﾞｰﾀ19段
ZR60793  ; C軸ﾜｰｸ曲げﾃﾞｰﾀ20段
ZR60795  ; C軸ﾜｰｸ曲げﾃﾞｰﾀ21段
ZR60797  ; C軸ﾜｰｸ曲げﾃﾞｰﾀ22段
ZR60799  ; C軸ﾜｰｸ曲げﾃﾞｰﾀ23段
ZR60801  ; C軸ﾜｰｸ曲げﾃﾞｰﾀ24段
ZR60803  ; C軸ﾜｰｸ曲げﾃﾞｰﾀ25段
ZR60805  ; C軸ﾜｰｸ曲げﾃﾞｰﾀ26段
ZR60807  ; C軸ﾜｰｸ曲げﾃﾞｰﾀ27段
ZR60809  ; C軸ﾜｰｸ曲げﾃﾞｰﾀ28段
ZR60811  ; C軸ﾜｰｸ曲げﾃﾞｰﾀ29段
ZR60813  ; C軸ﾜｰｸ曲げﾃﾞｰﾀ30段
W103  ; [CC-Link]ｸﾗﾝﾌﾟﾀﾞｲ一致出力ﾎﾟｲﾝﾄNO
W105  ; [CC-Link]ｸﾗﾝﾌﾟﾀﾞｲｻﾝﾌﾟﾘﾝｸﾞ/周期時
W106  ; [CC-Link]ｸﾗﾝﾌﾟﾀﾞｲ一致出力ﾎﾟｲﾝﾄNO
W10B  ; [CC-Link]ﾌﾟﾚｯｼｬﾀﾞｲ一致出力ﾎﾟｲﾝﾄN
W10D  ; [CC-Link]ﾌﾟﾚｯｼｬﾀﾞｲｻﾝﾌﾟﾘﾝｸﾞ/周期
W10E  ; [CC-Link]ﾌﾟﾚｯｼｬﾀﾞｲ一致出力ﾎﾟｲﾝﾄN
W113  ; [CC-Link]曲げ一致出力ﾎﾟｲﾝﾄNO.1設
W115  ; [CC-Link]曲げｻﾝﾌﾟﾘﾝｸﾞ/周期時間設
W116  ; [CC-Link]曲げ一致出力ﾎﾟｲﾝﾄNO.2設
W11B  ; [CC-Link]ﾍﾞﾝﾄﾞﾍｯﾄﾞｼﾌﾄ一致出力ﾎﾟｲ
W11D  ; [CC-Link]ﾍﾞﾝﾄﾞﾍｯﾄﾞｼﾌﾄｻﾝﾌﾟﾘﾝｸﾞ/周
W11E  ; [CC-Link]ﾍﾞﾝﾄﾞﾍｯﾄﾞｼﾌﾄ一致出力ﾎﾟｲ
W123  ; [CC-Link]ﾋﾈﾘ一致出力ﾎﾟｲﾝﾄNO.1設
W125  ; [CC-Link]ﾋﾈﾘｻﾝﾌﾟﾘﾝｸﾞ/周期時間設
W126  ; [CC-Link]ﾋﾈﾘ一致出力ﾎﾟｲﾝﾄNO.2設
W12B  ; [CC-Link]ﾁｬｯｸ開閉一致出力ﾎﾟｲﾝﾄNO
W12D  ; [CC-Link]ﾁｬｯｸ開閉ｻﾝﾌﾟﾘﾝｸﾞ/周期時
W12E  ; [CC-Link]ﾁｬｯｸ開閉一致出力ﾎﾟｲﾝﾄNO
W144  ; [CC-Link]IRDMVA1ｺﾝﾄﾛｰﾙﾌﾗｸﾞ0
W145  ; [CC-Link]IRDMVA1ｺﾝﾄﾛｰﾙﾌﾗｸﾞ2
W148  ; [CC-Link]IRDMVA2ｺﾝﾄﾛｰﾙﾌﾗｸﾞ0
W149  ; [CC-Link]IRDMVA2ｺﾝﾄﾛｰﾙﾌﾗｸﾞ2
W14C  ; [CC-Link]IRDMVA3ｺﾝﾄﾛｰﾙﾌﾗｸﾞ0
W14D  ; [CC-Link]IRDMVA3ｺﾝﾄﾛｰﾙﾌﾗｸﾞ2
W150  ; [CC-Link]IRDMAOｺﾝﾄﾛｰﾙﾌﾗｸﾞ0
W151  ; [CC-Link]IRDMAOｺﾝﾄﾛｰﾙﾌﾗｸﾞ2
W186  ; [CC-Link]IRDMCCLﾃﾞｰﾀ領域1
W190  ; [CC-Link]IRDMVA1ｺﾝﾄﾛｰﾙﾌﾗｸﾞ0
W191  ; [CC-Link]IRDMVA1ｺﾝﾄﾛｰﾙﾌﾗｸﾞ2
W194  ; [CC-Link]IRDMVA2ｺﾝﾄﾛｰﾙﾌﾗｸﾞ0
W195  ; [CC-Link]IRDMVA2ｺﾝﾄﾛｰﾙﾌﾗｸﾞ2
W198  ; [CC-Link]IRDMVA3ｺﾝﾄﾛｰﾙﾌﾗｸﾞ0
W199  ; [CC-Link]IRDMVA3ｺﾝﾄﾛｰﾙﾌﾗｸﾞ2
W19C  ; [CC-Link]IRDMAOｺﾝﾄﾛｰﾙﾌﾗｸﾞ0
W19D  ; [CC-Link]IRDMAOｺﾝﾄﾛｰﾙﾌﾗｸﾞ2
W202  ; [CC-Link]ｸﾗﾝﾌﾟﾀﾞｲﾗｯﾁｶｳﾝﾄ値/ｻﾝﾌﾟﾘ
W204  ; [CC-Link]ｸﾗﾝﾌﾟﾀﾞｲ周期ﾊﾟﾙｽｶｳﾝﾄ今
W20A  ; [CC-Link]ﾌﾟﾚｯｼｬﾀﾞｲﾗｯﾁｶｳﾝﾄ値/ｻﾝﾌﾟ
W20C  ; [CC-Link]ﾌﾟﾚｯｼｬﾀﾞｲ周期ﾊﾟﾙｽｶｳﾝﾄ今
W212  ; [CC-Link]曲げﾗｯﾁｶｳﾝﾄ値/ｻﾝﾌﾟﾘﾝｸﾞｶ
W214  ; [CC-Link]曲げ周期ﾊﾟﾙｽｶｳﾝﾄ今回値
W21A  ; [CC-Link]ﾍﾞﾝﾄﾞﾍｯﾄﾞｼﾌﾄﾗｯﾁｶｳﾝﾄ値/ｻ
W21C  ; [CC-Link]ﾍﾞﾝﾄﾞﾍｯﾄﾞｼﾌﾄ周期ﾊﾟﾙｽｶｳﾝ
W222  ; [CC-Link]ﾋﾈﾘﾗｯﾁｶｳﾝﾄ値/ｻﾝﾌﾟﾘﾝｸﾞｶｳ
W224  ; [CC-Link]ﾋﾈﾘ周期ﾊﾟﾙｽｶｳﾝﾄ今回値格
W22A  ; [CC-Link]ﾁｬｯｸ開閉ﾗｯﾁｶｳﾝﾄ値/ｻﾝﾌﾟﾘ
W22C  ; [CC-Link]ﾁｬｯｸ開閉周期ﾊﾟﾙｽｶｳﾝﾄ今
W244  ; [CC-Link]IRDMVA1ｽﾃｰﾀｽ
W246  ; [CC-Link]IRDMVA1出力電流値
W247  ; [CC-Link]IRDMVA1指令電流値
W248  ; [CC-Link]IRDMVA2ｽﾃｰﾀｽ
W24A  ; [CC-Link]IRDMVA2出力電流値
W24B  ; [CC-Link]IRDMVA2指令電流値
W24C  ; [CC-Link]IRDMVA3ｽﾃｰﾀｽ
W24E  ; [CC-Link]IRDMVA3出力電流値
W24F  ; [CC-Link]IRDMVA3指令電流値
W250  ; [CC-Link]IRDMAOｽﾃｰﾀｽﾌﾗｸﾞ0
W251  ; [CC-Link]IRDMAOｽﾃｰﾀｽﾌﾗｸﾞ2
W253  ; [CC-Link]IRDMAOｴﾗｰ/ｱﾗｰﾑ2
W286  ; [CC-Link]IRDMCCLﾃﾞｰﾀ領域1
W290  ; [CC-Link]IRDMVA1ｽﾃｰﾀｽ
W291  ; [CC-Link]IRDMVA1ｴﾗｰ/ｱﾗｰﾑ
W292  ; [CC-Link]IRDMVA1出力電流値
W293  ; [CC-Link]IRDMVA1指令電流値
W294  ; [CC-Link]IRDMVA2ｽﾃｰﾀｽ
W295  ; [CC-Link]IRDMVA2ｴﾗｰ/ｱﾗｰﾑ
W296  ; [CC-Link]IRDMVA2出力電流値
W297  ; [CC-Link]IRDMVA2指令電流値
W298  ; [CC-Link]IRDMVA3ｽﾃｰﾀｽ
W299  ; [CC-Link]IRDMVA3ｴﾗｰ/ｱﾗｰﾑ
W29A  ; [CC-Link]IRDMVA3出力電流値
W29B  ; [CC-Link]IRDMVA3指令電流値
W29C  ; [CC-Link]IRDMAOｽﾃｰﾀｽﾌﾗｸﾞ0
W29D  ; [CC-Link]IRDMAOｽﾃｰﾀｽﾌﾗｸﾞ2
W29E  ; [CC-Link]IRDMAOｴﾗｰ/ｱﾗｰﾑ0
W29F  ; [CC-Link]IRDMAOｴﾗｰ/ｱﾗｰﾑ2
W48A  ; 拡張 表示1行目
W48B  ; 手動ひねり 表示1行目
W48C  ; 空曲 表示1行目
W48D  ; 拡張 表示2行目
W48E  ; 手動ひねり 表示2行目
W48F  ; 空曲 表示2行目
W490  ; 拡張 表示3行目
W491  ; 手動ひねり 表示3行目
W492  ; 空曲 表示3行目
W493  ; 拡張 表示4行目
W494  ; 手動ひねり 表示4行目
W495  ; 空曲 表示4行目
W496  ; 拡張 表示5行目
W497  ; 手動ひねり 表示5行目
W498  ; 空曲 表示5行目
W499  ; 拡張 表示6行目
W49A  ; 手動ひねり 表示6行目
W49B  ; 空曲 表示6行目
W49C  ; 拡張 表示7行目
W49D  ; 手動ひねり 表示7行目
W49E  ; 空曲 表示7行目
W49F  ; 拡張 表示8行目
W4A0  ; 手動ひねり 表示8行目
W4A1  ; 空曲 表示8行目
W4A2  ; 拡張 表示9行目
W4A3  ; 手動ひねり 表示9行目
W4A4  ; 空曲 表示9行目
W4A5  ; 拡張 表示10行目
W4A6  ; 手動ひねり 表示10行目
W4A7  ; 空曲 表示10行目
W58A  ; SV1a_PB
W58B  ; SV1b_PB
W58C  ; SV2a_PB
W58D  ; SV3a_PB
W58E  ; SV4a_PB
W58F  ; SV4b_PB
W590  ; SV5a_PB
W591  ; SV5b_PB
W592  ; SV6a_PB
W593  ; SV6b_PB
W594  ; SV7a_PB
W595  ; SV7b_PB
W596  ; SV8a_PB
W597  ; SV8b_PB
W598  ; SV9a_PB
W599  ; SV9b_PB
W59A  ; SV10a_PB
W59B  ; SV10b_PB
W59C  ; SV11a_PB
W59D  ; SV11b_PB
W59E  ; SV12a_PB
W59F  ; SV12b_PB
W5A0  ; SV13a_PB
W5A1  ; SV13b_PB
W5A2  ; SV14a_PB
W5A3  ; SV14b_PB
W5A4  ; SV15a_PB
W5A5  ; SV15b_PB
W5A6  ; SV16a_PB
W5A7  ; SV16b_PB
W5A8  ; SV17a_PB
W5A9  ; SV17b_PB
W5AA  ; SV18a_PB
W5AB  ; SV18b_PB
W5AC  ; SV19a_PB
W5AD  ; SV19b_PB
W5AE  ; SV20a_PB
W5AF  ; SV20b_PB
W5B0  ; SV21a_PB
W5B1  ; SV21b_PB
W5B2  ; SV22a_PB
W5B3  ; SV22b_PB
W5B4  ; SV23a_PB
W5B5  ; SV23b_PB
W5B6  ; SV24a_PB
W5B7  ; SV24b_PB
W5B8  ; SV25a_PB
W5B9  ; SV25b_PB
W5BA  ; SV26a_PB
W5BB  ; SV26b_PB
W5BC  ; SV27a_PB
W5BD  ; SV27b_PB
W5BE  ; SV28a_PB
W5BF  ; SV28b_PB
W5C0  ; SV29a_PB
W5C1  ; SV29b_PB
W5C2  ; SV30a_PB
W5C3  ; SV30b_PB
W5C4  ; SV31a_PB
W5C5  ; SV31b_PB
W5C6  ; SV32a_PB
W5C7  ; SV32b_PB
W5C8  ; SV33a_PB
W5C9  ; SV33b_PB
W5CA  ; SV34a_PB
W5CB  ; SV34b_PB
W5CC  ; SV35a_PB
W5CD  ; SV35b_PB
W5CE  ; SV36a_PB
W5CF  ; SV36b_PB
W5D0  ; SV37a_PB
W5D1  ; SV37b_PB
W5D2  ; SV38a_PB
W5D3  ; SV38b_PB
W5D4  ; SV39a_PB
W5D5  ; SV39b_PB
W5D6  ; SV40a_PB
W5D7  ; SV40b_PB
W5DA  ; PV1_PB
W5DB  ; PV2_PB
W5DC  ; PV3_PB
W5DD  ; PV4_PB
W5DE  ; PV5_PB
W5DF  ; PV6_PB
W5E0  ; PV7_PB
W5E1  ; SE1_PB
W5E2  ; SE2_PB
W60A  ; (手割込)ｺﾚｯﾄﾁｬｯｸ_INL
W60B  ; (手割込)送り_INL
W60C  ; ｸﾗﾝﾌﾟ_INL
W60D  ; ﾌﾟﾚｯｼｬｰ_INL
W60E  ; ｻｲﾄﾞﾌﾞｰｽﾀｰ_INL
W60F  ; 曲げ_INL
W610  ; ﾍｯﾄﾞ昇降_INL
W611  ; ﾍｯﾄﾞｼﾌﾄ_INL
W612  ; ﾍｯﾄﾞｼﾌﾄ(左)_INL
W613  ; ﾍｯﾄﾞｼﾌﾄ(右)_INL
W614  ; 送り_INL
W615  ; ｺﾚｯﾄﾁｬｯｸ_INL
W616  ; ｾﾝﾀﾘﾝｸﾞ_INL
W617  ; 昇降ﾛｰﾗ_INL
W618  ; ﾌﾞｰｽﾄﾁｬｯｸ_INL
W619  ; ﾊﾞｯｸﾌﾞｰｽﾀ_INL
W61A  ; ﾌﾞｰｽﾀｰ受け_INL
W61B  ; NO.1ﾁｭｰﾌﾞ位置決めﾛｰﾗ_INL
W61C  ; ひねり_INL
W61D  ; NO.2ﾁｭｰﾌﾞ位置決めﾛｰﾗ_INL
W61E  ; ﾁｭｰﾌﾞ拡張_INL
W61F  ; NO.1ﾁｭｰﾌﾞｻﾎﾟｰﾄ_INL
W620  ; NO.2ﾁｭｰﾌﾞｻﾎﾟｰﾄ_INL
W621  ; NO.3ﾁｭｰﾌﾞｻﾎﾟｰﾄ_INL
W622  ; NO.4ﾁｭｰﾌﾞｻﾎﾟｰﾄ_INL
W623  ; ﾘﾄﾗｸﾄﾜｲﾊﾟｰ_INL
W624  ; ﾘﾄﾗｸﾄﾜｲﾊﾟｰｼﾌﾄ_INL
W625  ; ﾘﾄﾗｸﾄｼﾌﾄ_INL
W626  ; ﾘﾄﾗｸﾄﾜｲﾊﾟｰ注油_INL
W0E92  ; SV1a_LMP
W0E93  ; SV1b_LMP
W0E94  ; SV2a_LMP
W0E95  ; SV3a_LMP
W0E96  ; SV4a_LMP
W0E97  ; SV4b_LMP
W0E98  ; SV5a_LMP
W0E99  ; SV5b_LMP
W0E9A  ; SV6a_LMP
W0E9B  ; SV6b_LMP
W0E9C  ; SV7a_LMP
W0E9D  ; SV7b_LMP
W0E9E  ; SV8a_LMP
W0E9F  ; SV8b_LMP
W0EA0  ; SV9a_LMP
W0EA1  ; SV9b_LMP
W0EA2  ; SV10a_LMP
W0EA3  ; SV10b_LMP
W0EA4  ; SV11a_LMP
W0EA5  ; SV11b_LMP
W0EA6  ; SV12a_LMP
W0EA7  ; SV12b_LMP
W0EA8  ; SV13a_LMP
W0EA9  ; SV13b_LMP
W0EAA  ; SV14a_LMP
W0EAB  ; SV14b_LMP
W0EAC  ; SV15a_LMP
W0EAD  ; SV15b_LMP
W0EAE  ; SV16a_LMP
W0EAF  ; SV16b_LMP
W0EB0  ; SV17a_LMP
W0EB1  ; SV17b_LMP
W0EB2  ; SV18a_LMP
W0EB3  ; SV18b_LMP
W0EB4  ; SV19a_LMP
W0EB5  ; SV19b_LMP
W0EB6  ; SV20a_LMP
W0EB7  ; SV20b_LMP
W0EB8  ; SV21a_LMP
W0EB9  ; SV21b_LMP
W0EBA  ; SV22a_LMP
W0EBB  ; SV22b_LMP
W0EBC  ; SV23a_LMP
W0EBD  ; SV23b_LMP
W0EBE  ; SV24a_LMP
W0EBF  ; SV24b_LMP
W0EC0  ; SV25a_LMP
W0EC1  ; SV25b_LMP
W0EC2  ; SV26a_LMP
W0EC3  ; SV26b_LMP
W0EC4  ; SV27a_LMP
W0EC5  ; SV27b_LMP
W0EC6  ; SV28a_LMP
W0EC7  ; SV28b_LMP
W0EC8  ; SV29a_LMP
W0EC9  ; SV29b_LMP
W0ECA  ; SV30a_LMP
W0ECB  ; SV30b_LMP
W0ECC  ; SV31a_LMP
W0ECD  ; SV31b_LMP
W0ECE  ; SV32a_LMP
W0ECF  ; SV32b_LMP
W0ED0  ; SV33a_LMP
W0ED1  ; SV33b_LMP
W0ED2  ; SV34a_LMP
W0ED3  ; SV34b_LMP
W0ED4  ; SV35a_LMP
W0ED5  ; SV35b_LMP
W0ED6  ; SV36a_LMP
W0ED7  ; SV36b_LMP
W0ED8  ; SV37a_LMP
W0ED9  ; SV37b_LMP
W0EDA  ; SV38a_LMP
W0EDB  ; SV38b_LMP
W0EDC  ; SV39a_LMP
W0EDD  ; SV39b_LMP
W0EDE  ; SV40a_LMP
W0EDF  ; SV40b_LMP
T7  ; ﾜｰｸﾃﾞｰﾀ有ONﾃﾞｨﾚｰ
T11  ; 送りｻｰﾎﾞON出力後遅延
T16  ; 送り速度制御選択完了
T17  ; 送り速度制御選択遅延
T18  ; 送りﾄﾙｸ切替遅延
T19  ; 送り追従制御切替遅延
T36  ; 曲げ圧抜き確認
T106  ; 芯金圧抜き確認
T158  ; ﾜｲﾊﾟｰ注油間欠吐出/待ち時間
T159  ; ﾜｲﾊﾟｰ注油注油時間
T216  ; ﾘﾄﾗｸﾄﾌﾟﾚｯｼｬ位置決め手動後退時間
T247  ; 省略手動選択ﾀｲﾏｰ
T251  ; 曲げ時ﾌﾟﾚｯｼｬ開ﾃﾞｨﾚｰ
T252  ; 自動芯金ﾊｰﾌ遅延
T253  ; 端面検出後退開始遅延
T270  ; D70=060 ﾁｬｯｸ開時間
T280  ; D70=060 ﾁｬｯｸ開時間
T281  ; D70=210 ﾁｬｯｸ開時間
T282  ; 送りﾊﾞｯﾃﾘ低下
T291  ; ﾃﾞｰﾀ検索遅延
T300  ; W50_ﾃﾞｰﾀ保管表示遅延
C75  ; 曲げ    送り追従停止遅延
P100  ; 定義ｺｲﾙ
P201  ; 送り状態
P202  ; ﾋﾈﾘ状態
P203  ; 曲げ状態
P204  ; ｸﾗﾝﾌﾟﾀﾞｲ移動状態
P205  ; ﾌﾟﾚｯｼｬｰﾀﾞｲ移動状態
P206  ; ﾍｯﾄﾞｼﾌﾄ状態
P207  ; ｸﾗﾝﾌﾟ状態
P208  ; ﾌﾟﾚｯｼｬｰ状態
P209  ; ﾁｬｯｸ状態
P210  ; 芯金状態
P211  ; 状態
P212  ; 状態
P213  ; ﾊﾟｲﾌﾟ受け状態
P214  ; ﾌﾗﾝｼﾞ穴検出状態
P300  ; 異常ﾘｾｯﾄ
P301  ; 軽故障＿表示のみ
P302  ; 中故障　(停止)
P304  ; 重故障　(停止)
P305  ; 中故障　動作異常(一停)
P307  ; 故障のまとめ
P308  ; 故障追加発生
P400  ; 電源投入
P401  ; 油圧ﾎﾟﾝﾌﾟ運転
P402  ; 手動/自動運転準備OK
P410  ; ｽｷｬﾝﾀｲﾑ検出
P411  ; 表示中ﾍﾞｰｽ画面番号
P412  ; 表示中ｳｨﾝﾄﾞｳ画面番号
P413  ; ｽﾃｯﾌﾟﾓｰﾄﾞ
P420  ; ｽﾃｯﾌﾟ段数
P422  ; 送り長不足&干渉警報
P423  ; 自動定義
P424  ; 運転ﾓｰﾄﾞ
P425  ; ﾊﾟｲﾌﾟ選択
P426  ; ﾊﾟｲﾌﾟ抜き量
P427  ; ﾌﾗﾝｼﾞ穴検下降停止遅延時間
P430  ; 設定目標値
P431  ; 設定速度
P600  ; 原点復帰
P601  ; **原点復帰ｽﾃｯﾌﾟ
P700  ; 自動条件
P701  ; 自動運転
P704  ; 自動中ﾊﾟｲﾌﾟ抜き
P705  ; 自動中ｷｬﾚｯｼﾞ退避
P707  ; 短管曲げ条件
P708  ; 短管曲げ運転
P800  ; 自動準備条件定義
P801  ; 自動準備
P802  ; 自動準備ｽﾃｯﾌﾟ
P1100  ; ｸﾗﾝﾌﾟﾀﾞｲ手動前進
P1101  ; ｸﾗﾝﾌﾟﾀﾞｲ手動後退
P1102  ; ﾌﾟﾚｯｼｬｰﾀﾞｲ手動前進
P1103  ; ﾌﾟﾚｯｼｬｰﾀﾞｲ手動後退
P1106  ; ﾍｯﾄﾞｼﾌﾄR大
P1107  ; ﾍｯﾄﾞｼﾌﾄR小
P1108  ; ﾍｯﾄﾞｼﾌﾄ移動動作
P1213  ; **端面検出ｽﾃｯﾌﾟ
P1300  ; 捻り目標値
P1301  ; 捻り目標値到達
P1302  ; 捻り正転
P1303  ; 捻り逆転
P1306  ; 捻りﾌﾞﾚｰｷ解除
P1307  ; 捻り減速指令
P1580  ; ﾃﾞｰﾀ消去
P1600  ; 曲げ目標値
P1601  ; 曲げ目標値到達
P1602  ; 曲げ手動曲げ
P1603  ; 曲げ手動戻り
P1604  ; 曲げ指令ﾙｰﾁﾝ
P1605  ; 曲げ戻り指令
P1610  ; 曲げ速度設定
P1611  ; 曲げ速度加減速
P1612  ; 曲げｱﾅﾛｸﾞ出力
P1615  ; 送りﾄﾙｸ制限ｱﾅﾛｸﾞ出力
P1800  ; 送り目標値
P1802  ; 送り手動前進
P1803  ; 送り手動後退
P1810  ; 送りｻｰﾎﾞON
P1811  ; 送り運転指令まとめ
P1812  ; 送り停止
P1813  ; 送り追従ﾄﾙｸ制限
P1815  ; 送り送り量
P1816  ; 送り速度設定
P1818  ; 送り位置決め起動
P1819  ; 送り位置決めﾊﾟﾗﾒｰﾀ
P1821  ; 送り位置決めﾌﾟﾛｸﾞﾗﾑ起動
P1822  ; 送り原点復帰ﾌﾟﾛｸﾞﾗﾑ起動
P1840  ; FEED_ SERVO  ON
P1841  ; FEED_運転指令まとめ
P1842  ; FEED_停止
P1843  ; FEED_ﾄﾙｸ出力値
P1844  ; FEED_目標値
P1845  ; FEED_送り量
P1846  ; FEED_速度設定
P1847  ; FEED_速度制御ﾃﾞｰﾀ
P1848  ; FEED_位置決め起動
P1849  ; FEED_位置決めﾊﾟﾗﾒｰﾀ
P1900  ; 送り    ｻｰﾎﾞON
P1901  ; ACｻｰﾎﾞ異常ﾘｾｯﾄ
P1902  ; 基本ﾊﾟﾗﾒｰﾀ1設定
P1903  ; 基本ﾊﾟﾗﾒｰﾀ2設定
P1904  ; 詳細ﾊﾟﾗﾒｰﾀ2
P1905  ; 原点復帰基本ﾊﾟﾗﾒｰﾀ設定
P1906  ; 原点復帰詳細ﾊﾟﾗﾒｰﾀ設定
P1907  ; ｻｰﾎﾞﾊﾟﾗﾒｰﾀ
P2500  ; 曲げ完了表示検索
P2510  ; ﾊﾟｿｺﾝ立ち上がり確認
P2600  ; ﾘﾓｰﾄﾃﾞｰﾀ編集ﾙｰﾁﾝ呼出
P2602  ; B056画面初期値
P2611  ; *B055画面表示ﾙｰﾁﾝ
P2612  ; *B056画面表示ﾙｰﾁﾝ
P2613  ; *B057画面表示ﾙｰﾁﾝ
P2614  ; *ﾊﾟｲﾌﾟ抜き量&穴検補正ﾙｰﾁﾝ
P2800  ; ﾃﾞｰﾀ計算&検索
P2817  ; 現在段数表示ﾙｰﾁﾝ
P2900  ; 強制出力OFF
P2906  ; 芯金微調整
P2911  ; 芯金横移動
P2912  ; 芯金受け
P2914  ; ﾌﾗﾝｼﾞ穴検
P2920  ; Q64DA初期設定
P2921  ; PV2出力
P2923  ; PV2設定値*圧力比率
P2924  ; PV2出力補正
P2925  ; PV2ｱﾅﾛｸﾞ出力
P2931  ; PV3出力
P2932  ; PV3設定値
P2933  ; PV3設定値*圧力比率
P2934  ; PV3出力補正
P2935  ; PV3ｱﾅﾛｸﾞ出力
P2941  ; PV4出力
P2942  ; PV4設定値
P2943  ; PV4設定値*圧力比率
P2944  ; PV4出力補正
P2945  ; PV4ｱﾅﾛｸﾞ出力
P2960  ; IRDM-VA1初期設定
P2970  ; IRDM-VA2初期設定
P2980  ; IRDM-VA3初期設定
P3000  ; 画面切り替え
P3002  ; 自動運転中画面切換
P3003  ; ｳｲﾝﾄﾞｳ切替
P3005  ; ﾛｰｶﾙ/ﾘﾓｰﾄﾃﾞｰﾀ切替
P3010  ; ﾀｯﾁﾊﾟﾈﾙﾗﾝﾌﾟ表示
P3011  ; TP自動進行表示
P3012  ; ﾊﾟﾄﾗｲﾄ出力
P3013  ; 操作盤ﾗﾝﾌﾟ表示
P3014  ; 時刻設定
